LIN {X 0,Y 411.212,Z 369.263,A -85,B 0,C 180,E1 -10675.122,E2 -10675.122} C_VEL
LIN {X 0,Y 411.168,Z 369.267,A -85,B 0,C 180,E1 -10678.003,E2 -10678.003} C_VEL
LIN {X 0,Y 411.22,Z 369.26,A -85,B 0,C 180,E1 -10681.41,E2 -10681.41} C_VEL
LIN {X 0,Y 411.24,Z 369.258,A -85,B 0,C 180,E1 -10683.619,E2 -10683.619} C_VEL
LIN {X 0,Y 411.205,Z 369.264,A -85,B 0,C 180,E1 -10686.853,E2 -10686.853} C_VEL
LIN {X 0,Y 411.267,Z 369.256,A -85,B 0,C 180,E1 -10690.031,E2 -10690.031} C_VEL
LIN {X 0,Y 411.267,Z 369.255,A -85,B 0,C 180,E1 -10693.131,E2 -10693.131} C_VEL
LIN {X 0,Y 411.308,Z 369.251,A -85,B 0,C 180,E1 -10696.896,E2 -10696.896} C_VEL
LIN {X 0,Y 411.307,Z 369.253,A -85,B 0,C 180,E1 -10700.162,E2 -10700.162} C_VEL
LIN {X 0,Y 411.455,Z 369.23,A -85,B 0,C 180,E1 -10703.133,E2 -10703.133} C_VEL
LIN {X 0,Y 411.313,Z 369.249,A -85,B 0,C 180,E1 -10705.099,E2 -10705.099} C_VEL
LIN {X 0,Y 411.515,Z 369.226,A -85,B 0,C 180,E1 -10708.043,E2 -10708.043} C_VEL
LIN {X 0,Y 411.646,Z 369.21,A -85,B 0,C 180,E1 -10710,E2 -10710} C_VEL
LIN {X 0,Y 411.461,Z 369.229,A -85,B 0,C 180,E1 -10712.937,E2 -10712.937} C_VEL
LIN {X 0,Y 411.455,Z 369.232,A -85,B 0,C 180,E1 -10716.867,E2 -10716.867} C_VEL
LIN {X 0,Y 411.297,Z 369.253,A -85,B 0,C 180,E1 -10719.839,E2 -10719.839} C_VEL
LIN {X 0,Y 411.287,Z 369.252,A -85,B 0,C 180,E1 -10723.319,E2 -10723.319} C_VEL
LIN {X 0,Y 411.26,Z 369.256,A -85,B 0,C 180,E1 -10726.889,E2 -10726.889} C_VEL
LIN {X 0,Y 411.243,Z 369.257,A -85,B 0,C 180,E1 -10727.585,E2 -10727.585} C_VEL
LIN {X 0,Y 410.582,Z 369.343,A -85,B 0,C 180,E1 -10728.403,E2 -10728.403} C_VEL
LIN {X 0,Y 407.695,Z 369.704,A -85,B 0,C 180,E1 -10729.731,E2 -10729.731} C_VEL
LIN {X 0,Y 405.251,Z 370.006,A -85,B 0,C 180,E1 -10730.804,E2 -10730.804} C_VEL
LIN {X 0,Y 404.215,Z 370.136,A -85,B 0,C 180,E1 -10731.634,E2 -10731.634} C_VEL
LIN {X 0,Y 404.139,Z 370.141,A -85,B 0,C 180,E1 -10731.915,E2 -10731.915} C_VEL
LIN {X 0,Y 404.219,Z 370.134,A -85,B 0,C 180,E1 -10735.297,E2 -10735.297} C_VEL
LIN {X 0,Y 404.198,Z 370.137,A -85,B 0,C 180,E1 -10738,E2 -10738} C_VEL
LIN {X 0,Y 404.142,Z 370.145,A -85,B 0,C 180,E1 -10741.558,E2 -10741.558} C_VEL
LIN {X 0,Y 404.187,Z 370.137,A -85,B 0,C 180,E1 -10745.016,E2 -10745.016} C_VEL
LIN {X 0,Y 404.159,Z 370.141,A -85,B 0,C 180,E1 -10748.757,E2 -10748.757} C_VEL
LIN {X 0,Y 404.127,Z 370.147,A -85,B 0,C 180,E1 -10751.6,E2 -10751.6} C_VEL
LIN {X 0,Y 404.151,Z 370.141,A -85,B 0,C 180,E1 -10754.523,E2 -10754.523} C_VEL
LIN {X 0,Y 404.139,Z 370.146,A -85,B 0,C 180,E1 -10757.296,E2 -10757.296} C_VEL
LIN {X 0,Y 404.172,Z 370.139,A -85,B 0,C 180,E1 -10759.955,E2 -10759.955} C_VEL
LIN {X 0,Y 404.143,Z 370.144,A -85,B 0,C 180,E1 -10763.124,E2 -10763.124} C_VEL
LIN {X 0,Y 404.149,Z 370.141,A -85,B 0,C 180,E1 -10766.188,E2 -10766.188} C_VEL
LIN {X 0,Y 404.345,Z 370.296,A -85,B 0,C 180,E1 -10769.153,E2 -10769.153} C_VEL
LIN {X 0,Y 404.32,Z 374.446,A -85,B 0,C 180,E1 -10771.444,E2 -10771.444} C_VEL
LIN {X 0,Y 404.015,Z 380.585,A -85,B 0,C 180,E1 -10774.765,E2 -10774.765} C_VEL
LIN {X 0,Y 403.792,Z 386.695,A -85,B 0,C 180,E1 -10778.025,E2 -10778.025} C_VEL
LIN {X 0,Y 403.633,Z 392.803,A -85,B 0,C 180,E1 -10781.209,E2 -10781.209} C_VEL
LIN {X 0,Y 403.511,Z 398.878,A -85,B 0,C 180,E1 -10784.338,E2 -10784.338} C_VEL
LIN {X 0,Y 403.32,Z 405.986,A -85,B 0,C 180,E1 -10787.93,E2 -10787.93} C_VEL
LIN {X 0,Y 403.258,Z 409.014,A -85,B 0,C 180,E1 -10789.424,E2 -10789.424} C_VEL
LIN {X 0,Y 404.669,Z 419.398,A -85,B 0,C 180,E1 -10789.999,E2 -10789.999} C_VEL
LIN {X 0,Y 405.097,Z 425.037,A -85,B 0,C 180,E1 -10790.387,E2 -10790.387} C_VEL
LIN {X 0,Y 404.722,Z 435.358,A -85,B 0,C 180,E1 -10791.26,E2 -10791.26} C_VEL
LIN {X 0,Y 404.281,Z 444.367,A -85,B 0,C 180,E1 -10792.261,E2 -10792.261} C_VEL
LIN {X 0,Y 404.112,Z 451.373,A -85,B 0,C 180,E1 -10793.258,E2 -10793.258} C_VEL
LIN {X 0,Y 403.938,Z 458.258,A -85,B 0,C 180,E1 -10794.509,E2 -10794.509} C_VEL
LIN {X 0,Y 403.774,Z 462.57,A -85,B 0,C 180,E1 -10795.508,E2 -10795.508} C_VEL
LIN {X 0,Y 403.609,Z 465.969,A -85,B 0,C 180,E1 -10796.506,E2 -10796.506} C_VEL
LIN {X 0,Y 403.281,Z 469.606,A -85,B 0,C 180,E1 -10798.003,E2 -10798.003} C_VEL
LIN {X 0,Y 403.192,Z 471.134,A -85,B 0,C 180,E1 -10799.001,E2 -10799.001} C_VEL
LIN {X 0,Y 403.19,Z 471.985,A -85,B 0,C 180,E1 -10800,E2 -10800} C_VEL
LIN {X 0,Y 403.247,Z 472.168,A -85,B 0,C 180,E1 -10800.999,E2 -10800.999} C_VEL
LIN {X 0,Y 403.356,Z 471.686,A -85,B 0,C 180,E1 -10801.997,E2 -10801.997} C_VEL
LIN {X 0,Y 403.54,Z 470.533,A -85,B 0,C 180,E1 -10802.995,E2 -10802.995} C_VEL
LIN {X 0,Y 404.138,Z 467.465,A -85,B 0,C 180,E1 -10804.488,E2 -10804.488} C_VEL
LIN {X 0,Y 404.326,Z 464.514,A -85,B 0,C 180,E1 -10805.486,E2 -10805.486} C_VEL
LIN {X 0,Y 404.807,Z 459.63,A -85,B 0,C 180,E1 -10806.73,E2 -10806.73} C_VEL
LIN {X 0,Y 405.372,Z 453.215,A -85,B 0,C 180,E1 -10807.972,E2 -10807.972} C_VEL
LIN {X 0,Y 405.95,Z 446.675,A -85,B 0,C 180,E1 -10808.964,E2 -10808.964} C_VEL
LIN {X 0,Y 406.576,Z 438.47,A -85,B 0,C 180,E1 -10809.954,E2 -10809.954} C_VEL
LIN {X 0,Y 407.173,Z 429.296,A -85,B 0,C 180,E1 -10810.819,E2 -10810.819} C_VEL
LIN {X 0,Y 406.43,Z 423.17,A -85,B 0,C 180,E1 -10811.344,E2 -10811.344} C_VEL
LIN {X 0,Y 404.018,Z 412.539,A -85,B 0,C 180,E1 -10812.176,E2 -10812.176} C_VEL
LIN {X 0,Y 404.254,Z 407.353,A -85,B 0,C 180,E1 -10815.116,E2 -10815.116} C_VEL
LIN {X 0,Y 404.598,Z 402.059,A -85,B 0,C 180,E1 -10818.22,E2 -10818.22} C_VEL
LIN {X 0,Y 404.945,Z 396.896,A -85,B 0,C 180,E1 -10821.375,E2 -10821.375} C_VEL
LIN {X 0,Y 405.44,Z 391.905,A -85,B 0,C 180,E1 -10824.584,E2 -10824.584} C_VEL
LIN {X 0,Y 406.072,Z 386.86,A -85,B 0,C 180,E1 -10828.033,E2 -10828.033} C_VEL
LIN {X 0,Y 406.384,Z 384.059,A -85,B 0,C 180,E1 -10830.151,E2 -10830.151} C_VEL
LIN {X 0,Y 406.317,Z 381.396,A -85,B 0,C 180,E1 -10832.426,E2 -10832.426} C_VEL
LIN {X 0,Y 406.022,Z 379.03,A -85,B 0,C 180,E1 -10834.835,E2 -10834.835} C_VEL
LIN {X 0,Y 405.683,Z 377.136,A -85,B 0,C 180,E1 -10837.325,E2 -10837.325} C_VEL
LIN {X 0,Y 405.446,Z 375.637,A -85,B 0,C 180,E1 -10840.297,E2 -10840.297} C_VEL
LIN {X 0,Y 405.397,Z 375.192,A -85,B 0,C 180,E1 -10843.271,E2 -10843.271} C_VEL
LIN {X 0,Y 405.551,Z 375.903,A -85,B 0,C 180,E1 -10846.117,E2 -10846.117} C_VEL
LIN {X 0,Y 406.076,Z 377.767,A -85,B 0,C 180,E1 -10848.877,E2 -10848.877} C_VEL
LIN {X 0,Y 406.772,Z 380.667,A -85,B 0,C 180,E1 -10851.538,E2 -10851.538} C_VEL
LIN {X 0,Y 408.037,Z 385.656,A -85,B 0,C 180,E1 -10854.76,E2 -10854.76} C_VEL
LIN {X 0,Y 409.173,Z 390.814,A -85,B 0,C 180,E1 -10857.313,E2 -10857.313} C_VEL
LIN {X 0,Y 410.133,Z 396.458,A -85,B 0,C 180,E1 -10859.635,E2 -10859.635} C_VEL
LIN {X 0,Y 409.985,Z 399.501,A -85,B 0,C 180,E1 -10860.695,E2 -10860.695} C_VEL
LIN {X 0,Y 407.911,Z 410.385,A -85,B 0,C 180,E1 -10864.008,E2 -10864.008} C_VEL
LIN {X 0,Y 406.44,Z 421.407,A -85,B 0,C 180,E1 -10867.104,E2 -10867.104} C_VEL
LIN {X 0,Y 405.209,Z 434.333,A -85,B 0,C 180,E1 -10870.496,E2 -10870.496} C_VEL
LIN {X 0,Y 404.648,Z 442.082,A -85,B 0,C 180,E1 -10872.397,E2 -10872.397} C_VEL
LIN {X 0,Y 406.509,Z 454.809,A -85,B 0,C 180,E1 -10872.908,E2 -10872.908} C_VEL
LIN {X 0,Y 407.267,Z 468.253,A -85,B 0,C 180,E1 -10873.601,E2 -10873.601} C_VEL
LIN {X 0,Y 406.773,Z 479.668,A -85,B 0,C 180,E1 -10874.338,E2 -10874.338} C_VEL
LIN {X 0,Y 405.87,Z 491.757,A -85,B 0,C 180,E1 -10875.33,E2 -10875.33} C_VEL
LIN {X 0,Y 405.11,Z 502.511,A -85,B 0,C 180,E1 -10876.462,E2 -10876.462} C_VEL
LIN {X 0,Y 404.391,Z 512.142,A -85,B 0,C 180,E1 -10877.708,E2 -10877.708} C_VEL
LIN {X 0,Y 403.888,Z 520.09,A -85,B 0,C 180,E1 -10878.965,E2 -10878.965} C_VEL
LIN {X 0,Y 403.457,Z 527.841,A -85,B 0,C 180,E1 -10880.474,E2 -10880.474} C_VEL
LIN {X 0,Y 403.222,Z 534.087,A -85,B 0,C 180,E1 -10881.985,E2 -10881.985} C_VEL
LIN {X 0,Y 403.136,Z 539.248,A -85,B 0,C 180,E1 -10883.567,E2 -10883.567} C_VEL
LIN {X 0,Y 403.096,Z 542.795,A -85,B 0,C 180,E1 -10884.999,E2 -10884.999} C_VEL
LIN {X 0,Y 403.113,Z 544.709,A -85,B 0,C 180,E1 -10886.001,E2 -10886.001} C_VEL
LIN {X 0,Y 403.202,Z 546.163,A -85,B 0,C 180,E1 -10887.002,E2 -10887.002} C_VEL
LIN {X 0,Y 403.218,Z 547.195,A -85,B 0,C 180,E1 -10888.002,E2 -10888.002} C_VEL
LIN {X 0,Y 403.123,Z 547.774,A -85,B 0,C 180,E1 -10889.001,E2 -10889.001} C_VEL
LIN {X 0,Y 403.102,Z 547.905,A -85,B 0,C 180,E1 -10890,E2 -10890} C_VEL
LIN {X 0,Y 403.121,Z 547.631,A -85,B 0,C 180,E1 -10890.999,E2 -10890.999} C_VEL
LIN {X 0,Y 403.223,Z 546.941,A -85,B 0,C 180,E1 -10891.997,E2 -10891.997} C_VEL
LIN {X 0,Y 403.268,Z 545.766,A -85,B 0,C 180,E1 -10892.997,E2 -10892.997} C_VEL
LIN {X 0,Y 403.099,Z 543.145,A -85,B 0,C 180,E1 -10894.5,E2 -10894.5} C_VEL
LIN {X 0,Y 403.142,Z 539.441,A -85,B 0,C 180,E1 -10896.004,E2 -10896.004} C_VEL
LIN {X 0,Y 403.201,Z 534.528,A -85,B 0,C 180,E1 -10897.512,E2 -10897.512} C_VEL
LIN {X 0,Y 403.358,Z 528.258,A -85,B 0,C 180,E1 -10899.022,E2 -10899.022} C_VEL
LIN {X 0,Y 403.681,Z 520.298,A -85,B 0,C 180,E1 -10900.533,E2 -10900.533} C_VEL
LIN {X 0,Y 404.134,Z 512.119,A -85,B 0,C 180,E1 -10901.79,E2 -10901.79} C_VEL
LIN {X 0,Y 404.728,Z 502.074,A -85,B 0,C 180,E1 -10903.046,E2 -10903.046} C_VEL
LIN {X 0,Y 405.281,Z 492.039,A -85,B 0,C 180,E1 -10904.05,E2 -10904.05} C_VEL
LIN {X 0,Y 405.86,Z 481.103,A -85,B 0,C 180,E1 -10904.926,E2 -10904.926} C_VEL
LIN {X 0,Y 406.416,Z 468.992,A -85,B 0,C 180,E1 -10905.676,E2 -10905.676} C_VEL
LIN {X 0,Y 405.399,Z 456.125,A -85,B 0,C 180,E1 -10906.276,E2 -10906.276} C_VEL
LIN {X 0,Y 404.221,Z 443.249,A -85,B 0,C 180,E1 -10906.7,E2 -10906.7} C_VEL
LIN {X 0,Y 405.015,Z 430.654,A -85,B 0,C 180,E1 -10909.778,E2 -10909.778} C_VEL
LIN {X 0,Y 406.134,Z 416.925,A -85,B 0,C 180,E1 -10913.184,E2 -10913.184} C_VEL
LIN {X 0,Y 407.489,Z 403.197,A -85,B 0,C 180,E1 -10916.642,E2 -10916.642} C_VEL
LIN {X 0,Y 408.621,Z 392.664,A -85,B 0,C 180,E1 -10919.352,E2 -10919.352} C_VEL
LIN {X 0,Y 407.859,Z 387.494,A -85,B 0,C 180,E1 -10920.778,E2 -10920.778} C_VEL
LIN {X 0,Y 405.306,Z 375.4,A -85,B 0,C 180,E1 -10924.301,E2 -10924.301} C_VEL
LIN {X 0,Y 404.175,Z 370.14,A -85,B 0,C 180,E1 -10925.906,E2 -10925.906} C_VEL
LIN {X 0,Y 404.155,Z 370.141,A -85,B 0,C 180,E1 -10928.757,E2 -10928.757} C_VEL
LIN {X 0,Y 404.125,Z 370.148,A -85,B 0,C 180,E1 -10931.6,E2 -10931.6} C_VEL
LIN {X 0,Y 404.151,Z 370.143,A -85,B 0,C 180,E1 -10934.523,E2 -10934.523} C_VEL
LIN {X 0,Y 404.141,Z 370.142,A -85,B 0,C 180,E1 -10937.296,E2 -10937.296} C_VEL
LIN {X 0,Y 404.169,Z 370.141,A -85,B 0,C 180,E1 -10939.955,E2 -10939.955} C_VEL
LIN {X 0,Y 404.141,Z 370.142,A -85,B 0,C 180,E1 -10943.124,E2 -10943.124} C_VEL
LIN {X 0,Y 404.146,Z 370.144,A -85,B 0,C 180,E1 -10946.188,E2 -10946.188} C_VEL
LIN {X 0,Y 404.146,Z 370.143,A -85,B 0,C 180,E1 -10949.715,E2 -10949.715} C_VEL
LIN {X 0,Y 404.196,Z 370.135,A -85,B 0,C 180,E1 -10953.123,E2 -10953.123} C_VEL
LIN {X 0,Y 404.178,Z 370.139,A -85,B 0,C 180,E1 -10955.334,E2 -10955.334} C_VEL
LIN {X 0,Y 404.14,Z 370.143,A -85,B 0,C 180,E1 -10958.581,E2 -10958.581} C_VEL
LIN {X 0,Y 404.211,Z 370.137,A -85,B 0,C 180,E1 -10961.762,E2 -10961.762} C_VEL
LIN {X 0,Y 404.208,Z 370.134,A -85,B 0,C 180,E1 -10964.882,E2 -10964.882} C_VEL
LIN {X 0,Y 404.258,Z 370.13,A -85,B 0,C 180,E1 -10967.959,E2 -10967.959} C_VEL
LIN {X 0,Y 404.434,Z 370.106,A -85,B 0,C 180,E1 -10972.1,E2 -10972.1} C_VEL
LIN {X 0,Y 404.425,Z 370.108,A -85,B 0,C 180,E1 -10974.015,E2 -10974.015} C_VEL
LIN {X 0,Y 404.484,Z 370.102,A -85,B 0,C 180,E1 -10978.009,E2 -10978.009} C_VEL
LIN {X 0,Y 404.613,Z 370.085,A -85,B 0,C 180,E1 -10980,E2 -10980} C_VEL
LIN {X 0,Y 404.417,Z 370.108,A -85,B 0,C 180,E1 -10982.988,E2 -10982.988} C_VEL
LIN {X 0,Y 404.413,Z 370.11,A -85,B 0,C 180,E1 -10986.987,E2 -10986.987} C_VEL
LIN {X 0,Y 404.272,Z 370.127,A -85,B 0,C 180,E1 -10990.011,E2 -10990.011} C_VEL
LIN {X 0,Y 404.267,Z 370.129,A -85,B 0,C 180,E1 -10993.211,E2 -10993.211} C_VEL
LIN {X 0,Y 404.217,Z 370.136,A -85,B 0,C 180,E1 -10997.007,E2 -10997.007} C_VEL
LIN {X 0,Y 404.165,Z 370.14,A -85,B 0,C 180,E1 -11000.352,E2 -11000.352} C_VEL
LIN {X 0,Y 404.171,Z 370.14,A -85,B 0,C 180,E1 -11003.575,E2 -11003.575} C_VEL
LIN {X 0,Y 404.185,Z 370.136,A -85,B 0,C 180,E1 -11005.766,E2 -11005.766} C_VEL
LIN {X 0,Y 404.196,Z 370.135,A -85,B 0,C 180,E1 -11008,E2 -11008} C_VEL
LIN {X 0,Y 404.14,Z 370.144,A -85,B 0,C 180,E1 -11011.558,E2 -11011.558} C_VEL
LIN {X 0,Y 404.187,Z 370.14,A -85,B 0,C 180,E1 -11015.016,E2 -11015.016} C_VEL
LIN {X 0,Y 404.158,Z 370.145,A -85,B 0,C 180,E1 -11018.757,E2 -11018.757} C_VEL
LIN {X 0,Y 404.124,Z 370.145,A -85,B 0,C 180,E1 -11021.6,E2 -11021.6} C_VEL
LIN {X 0,Y 404.148,Z 370.143,A -85,B 0,C 180,E1 -11024.522,E2 -11024.522} C_VEL
LIN {X 0,Y 404.141,Z 370.142,A -85,B 0,C 180,E1 -11027.296,E2 -11027.296} C_VEL
LIN {X 0,Y 404.17,Z 370.138,A -85,B 0,C 180,E1 -11029.956,E2 -11029.956} C_VEL
LIN {X 0,Y 404.138,Z 370.145,A -85,B 0,C 180,E1 -11033.125,E2 -11033.125} C_VEL
LIN {X 0,Y 404.146,Z 370.143,A -85,B 0,C 180,E1 -11036.188,E2 -11036.188} C_VEL
LIN {X 0,Y 404.147,Z 370.14,A -85,B 0,C 180,E1 -11039.715,E2 -11039.715} C_VEL
LIN {X 0,Y 404.197,Z 370.136,A -85,B 0,C 180,E1 -11043.123,E2 -11043.123} C_VEL
LIN {X 0,Y 404.179,Z 370.138,A -85,B 0,C 180,E1 -11045.335,E2 -11045.335} C_VEL
LIN {X 0,Y 404.165,Z 370.143,A -85,B 0,C 180,E1 -11048.582,E2 -11048.582} C_VEL
LIN {X 0,Y 404.217,Z 370.133,A -85,B 0,C 180,E1 -11051.762,E2 -11051.762} C_VEL
LIN {X 0,Y 404.214,Z 370.134,A -85,B 0,C 180,E1 -11054.882,E2 -11054.882} C_VEL
LIN {X 0,Y 404.259,Z 370.129,A -85,B 0,C 180,E1 -11057.959,E2 -11057.959} C_VEL
LIN {X 0,Y 404.386,Z 370.115,A -85,B 0,C 180,E1 -11062.008,E2 -11062.008} C_VEL
LIN {X 0,Y 404.422,Z 370.111,A -85,B 0,C 180,E1 -11064.015,E2 -11064.015} C_VEL
LIN {X 0,Y 404.484,Z 370.102,A -85,B 0,C 180,E1 -11068.009,E2 -11068.009} C_VEL
LIN {X 0,Y 404.615,Z 370.086,A -85,B 0,C 180,E1 -11070,E2 -11070} C_VEL
LIN {X 0,Y 404.419,Z 370.106,A -85,B 0,C 180,E1 -11072.989,E2 -11072.989} C_VEL
LIN {X 0,Y 404.422,Z 370.109,A -85,B 0,C 180,E1 -11075.985,E2 -11075.985} C_VEL
LIN {X 0,Y 404.295,Z 370.124,A -85,B 0,C 180,E1 -11079.001,E2 -11079.001} C_VEL
LIN {X 0,Y 404.26,Z 370.13,A -85,B 0,C 180,E1 -11082.042,E2 -11082.042} C_VEL
LIN {X 0,Y 404.21,Z 370.134,A -85,B 0,C 180,E1 -11085.118,E2 -11085.118} C_VEL
LIN {X 0,Y 404.213,Z 370.135,A -85,B 0,C 180,E1 -11088.238,E2 -11088.238} C_VEL
LIN {X 0,Y 404.142,Z 370.144,A -85,B 0,C 180,E1 -11091.419,E2 -11091.419} C_VEL
LIN {X 0,Y 404.139,Z 370.141,A -85,B 0,C 180,E1 -11091.915,E2 -11091.915} C_VEL
LIN {X 0,Y 403.496,Z 370.223,A -85,B 0,C 180,E1 -11092.746,E2 -11092.746} C_VEL
LIN {X 0,Y 400.664,Z 370.576,A -85,B 0,C 180,E1 -11094.098,E2 -11094.098} C_VEL
LIN {X 0,Y 398.254,Z 370.877,A -85,B 0,C 180,E1 -11095.19,E2 -11095.19} C_VEL
LIN {X 0,Y 397.22,Z 371.005,A -85,B 0,C 180,E1 -11096.034,E2 -11096.034} C_VEL
LIN {X 0,Y 397.137,Z 371.014,A -85,B 0,C 180,E1 -11096.32,E2 -11096.32} C_VEL
LIN {X 0,Y 397.125,Z 371.016,A -85,B 0,C 180,E1 -11098.544,E2 -11098.544} C_VEL
LIN {X 0,Y 397.081,Z 371.023,A -85,B 0,C 180,E1 -11102.072,E2 -11102.072} C_VEL
LIN {X 0,Y 397.122,Z 371.02,A -85,B 0,C 180,E1 -11105.503,E2 -11105.503} C_VEL
LIN {X 0,Y 397.134,Z 371.017,A -85,B 0,C 180,E1 -11108.862,E2 -11108.862} C_VEL
LIN {X 0,Y 397.074,Z 371.023,A -85,B 0,C 180,E1 -11112.267,E2 -11112.267} C_VEL
LIN {X 0,Y 397.092,Z 371.022,A -85,B 0,C 180,E1 -11115.069,E2 -11115.069} C_VEL
LIN {X 0,Y 397.069,Z 371.022,A -85,B 0,C 180,E1 -11118.021,E2 -11118.021} C_VEL
LIN {X 0,Y 397.136,Z 371.017,A -85,B 0,C 180,E1 -11121.138,E2 -11121.138} C_VEL
LIN {X 0,Y 397.123,Z 371.017,A -85,B 0,C 180,E1 -11124.497,E2 -11124.497} C_VEL
LIN {X 0,Y 397.164,Z 371.013,A -85,B 0,C 180,E1 -11128.145,E2 -11128.145} C_VEL
LIN {X 0,Y 397.291,Z 371.125,A -85,B 0,C 180,E1 -11129.062,E2 -11129.062} C_VEL
LIN {X 0,Y 397.323,Z 374.396,A -85,B 0,C 180,E1 -11130.894,E2 -11130.894} C_VEL
LIN {X 0,Y 396.973,Z 381.037,A -85,B 0,C 180,E1 -11134.543,E2 -11134.543} C_VEL
LIN {X 0,Y 396.763,Z 386.773,A -85,B 0,C 180,E1 -11137.621,E2 -11137.621} C_VEL
LIN {X 0,Y 396.589,Z 392.898,A -85,B 0,C 180,E1 -11140.862,E2 -11140.862} C_VEL
LIN {X 0,Y 396.448,Z 399,A -85,B 0,C 180,E1 -11144.051,E2 -11144.051} C_VEL
LIN {X 0,Y 396.272,Z 406.161,A -85,B 0,C 180,E1 -11147.712,E2 -11147.712} C_VEL
LIN {X 0,Y 396.16,Z 409.279,A -85,B 0,C 180,E1 -11149.265,E2 -11149.265} C_VEL
LIN {X 0,Y 397.641,Z 420.176,A -85,B 0,C 180,E1 -11149.884,E2 -11149.884} C_VEL
LIN {X 0,Y 398.045,Z 426.586,A -85,B 0,C 180,E1 -11150.344,E2 -11150.344} C_VEL
LIN {X 0,Y 397.651,Z 436.659,A -85,B 0,C 180,E1 -11151.232,E2 -11151.232} C_VEL
LIN {X 0,Y 397.231,Z 445.211,A -85,B 0,C 180,E1 -11152.215,E2 -11152.215} C_VEL
LIN {X 0,Y 397.057,Z 453.143,A -85,B 0,C 180,E1 -11153.393,E2 -11153.393} C_VEL
LIN {X 0,Y 396.838,Z 459.749,A -85,B 0,C 180,E1 -11154.665,E2 -11154.665} C_VEL
LIN {X 0,Y 396.593,Z 464.783,A -85,B 0,C 180,E1 -11155.935,E2 -11155.935} C_VEL
LIN {X 0,Y 396.36,Z 467.853,A -85,B 0,C 180,E1 -11156.951,E2 -11156.951} C_VEL
LIN {X 0,Y 396.233,Z 470.158,A -85,B 0,C 180,E1 -11157.967,E2 -11157.967} C_VEL
LIN {X 0,Y 396.136,Z 471.757,A -85,B 0,C 180,E1 -11158.983,E2 -11158.983} C_VEL
LIN {X 0,Y 396.13,Z 472.676,A -85,B 0,C 180,E1 -11160,E2 -11160} C_VEL
LIN {X 0,Y 396.189,Z 472.923,A -85,B 0,C 180,E1 -11161.016,E2 -11161.016} C_VEL
LIN {X 0,Y 396.309,Z 472.502,A -85,B 0,C 180,E1 -11162.033,E2 -11162.033} C_VEL
LIN {X 0,Y 396.505,Z 471.41,A -85,B 0,C 180,E1 -11163.048,E2 -11163.048} C_VEL
LIN {X 0,Y 397.127,Z 468.457,A -85,B 0,C 180,E1 -11164.568,E2 -11164.568} C_VEL
LIN {X 0,Y 397.365,Z 465.61,A -85,B 0,C 180,E1 -11165.582,E2 -11165.582} C_VEL
LIN {X 0,Y 397.876,Z 460.871,A -85,B 0,C 180,E1 -11166.848,E2 -11166.848} C_VEL
LIN {X 0,Y 398.461,Z 454.631,A -85,B 0,C 180,E1 -11168.112,E2 -11168.112} C_VEL
LIN {X 0,Y 399.216,Z 446.466,A -85,B 0,C 180,E1 -11169.372,E2 -11169.372} C_VEL
LIN {X 0,Y 399.932,Z 438.019,A -85,B 0,C 180,E1 -11170.377,E2 -11170.377} C_VEL
LIN {X 0,Y 400.41,Z 428.651,A -85,B 0,C 180,E1 -11171.26,E2 -11171.26} C_VEL
LIN {X 0,Y 398.605,Z 419.229,A -85,B 0,C 180,E1 -11172.086,E2 -11172.086} C_VEL
LIN {X 0,Y 397.088,Z 413.056,A -85,B 0,C 180,E1 -11172.57,E2 -11172.57} C_VEL
LIN {X 0,Y 397.396,Z 406.452,A -85,B 0,C 180,E1 -11176.437,E2 -11176.437} C_VEL
LIN {X 0,Y 397.787,Z 401.229,A -85,B 0,C 180,E1 -11179.614,E2 -11179.614} C_VEL
LIN {X 0,Y 398.332,Z 395.288,A -85,B 0,C 180,E1 -11183.441,E2 -11183.441} C_VEL
LIN {X 0,Y 399.018,Z 389.746,A -85,B 0,C 180,E1 -11187.255,E2 -11187.255} C_VEL
LIN {X 0,Y 399.437,Z 386.761,A -85,B 0,C 180,E1 -11189.515,E2 -11189.515} C_VEL
LIN {X 0,Y 399.538,Z 383.439,A -85,B 0,C 180,E1 -11192.399,E2 -11192.399} C_VEL
LIN {X 0,Y 399.185,Z 380.624,A -85,B 0,C 180,E1 -11195.521,E2 -11195.521} C_VEL
LIN {X 0,Y 398.822,Z 378.445,A -85,B 0,C 180,E1 -11199.162,E2 -11199.162} C_VEL
LIN {X 0,Y 398.721,Z 377.703,A -85,B 0,C 180,E1 -11202.052,E2 -11202.052} C_VEL
LIN {X 0,Y 398.827,Z 378.008,A -85,B 0,C 180,E1 -11204.819,E2 -11204.819} C_VEL
LIN {X 0,Y 399.213,Z 379.398,A -85,B 0,C 180,E1 -11207.68,E2 -11207.68} C_VEL
LIN {X 0,Y 399.88,Z 382.14,A -85,B 0,C 180,E1 -11210.652,E2 -11210.652} C_VEL
LIN {X 0,Y 400.749,Z 385.848,A -85,B 0,C 180,E1 -11213.397,E2 -11213.397} C_VEL
LIN {X 0,Y 401.642,Z 389.151,A -85,B 0,C 180,E1 -11215.327,E2 -11215.327} C_VEL
LIN {X 0,Y 402.693,Z 394.363,A -85,B 0,C 180,E1 -11217.839,E2 -11217.839} C_VEL
LIN {X 0,Y 403.354,Z 398.737,A -85,B 0,C 180,E1 -11219.649,E2 -11219.649} C_VEL
LIN {X 0,Y 403.051,Z 401.938,A -85,B 0,C 180,E1 -11220.775,E2 -11220.775} C_VEL
LIN {X 0,Y 400.978,Z 412.337,A -85,B 0,C 180,E1 -11224.012,E2 -11224.012} C_VEL
LIN {X 0,Y 399.404,Z 423.52,A -85,B 0,C 180,E1 -11227.225,E2 -11227.225} C_VEL
LIN {X 0,Y 398.15,Z 436.391,A -85,B 0,C 180,E1 -11230.672,E2 -11230.672} C_VEL
LIN {X 0,Y 397.711,Z 441.528,A -85,B 0,C 180,E1 -11231.993,E2 -11231.993} C_VEL
LIN {X 0,Y 399.636,Z 454.304,A -85,B 0,C 180,E1 -11232.535,E2 -11232.535} C_VEL
LIN {X 0,Y 400.372,Z 467.262,A -85,B 0,C 180,E1 -11233.221,E2 -11233.221} C_VEL
LIN {X 0,Y 400.317,Z 474.503,A -85,B 0,C 180,E1 -11233.686,E2 -11233.686} C_VEL
LIN {X 0,Y 399.431,Z 486.15,A -85,B 0,C 180,E1 -11234.566,E2 -11234.566} C_VEL
LIN {X 0,Y 398.632,Z 496.658,A -85,B 0,C 180,E1 -11235.58,E2 -11235.58} C_VEL
LIN {X 0,Y 397.908,Z 506.32,A -85,B 0,C 180,E1 -11236.726,E2 -11236.726} C_VEL
LIN {X 0,Y 397.187,Z 515.15,A -85,B 0,C 180,E1 -11238,E2 -11238} C_VEL
LIN {X 0,Y 396.564,Z 523.737,A -85,B 0,C 180,E1 -11239.534,E2 -11239.534} C_VEL
LIN {X 0,Y 396.259,Z 530.655,A -85,B 0,C 180,E1 -11241.072,E2 -11241.072} C_VEL
LIN {X 0,Y 396.095,Z 536.981,A -85,B 0,C 180,E1 -11242.865,E2 -11242.865} C_VEL
LIN {X 0,Y 396.029,Z 541.076,A -85,B 0,C 180,E1 -11244.399,E2 -11244.399} C_VEL
LIN {X 0,Y 396.023,Z 544.085,A -85,B 0,C 180,E1 -11245.929,E2 -11245.929} C_VEL
LIN {X 0,Y 396.13,Z 545.524,A -85,B 0,C 180,E1 -11246.949,E2 -11246.949} C_VEL
LIN {X 0,Y 396.167,Z 546.542,A -85,B 0,C 180,E1 -11247.967,E2 -11247.967} C_VEL
LIN {X 0,Y 396.071,Z 547.083,A -85,B 0,C 180,E1 -11248.983,E2 -11248.983} C_VEL
LIN {X 0,Y 396.047,Z 547.197,A -85,B 0,C 180,E1 -11250,E2 -11250} C_VEL
LIN {X 0,Y 396.07,Z 546.905,A -85,B 0,C 180,E1 -11251.017,E2 -11251.017} C_VEL
LIN {X 0,Y 396.175,Z 546.172,A -85,B 0,C 180,E1 -11252.033,E2 -11252.033} C_VEL
LIN {X 0,Y 396.193,Z 544.97,A -85,B 0,C 180,E1 -11253.05,E2 -11253.05} C_VEL
LIN {X 0,Y 396.026,Z 542.296,A -85,B 0,C 180,E1 -11254.58,E2 -11254.58} C_VEL
LIN {X 0,Y 396.085,Z 538.534,A -85,B 0,C 180,E1 -11256.111,E2 -11256.111} C_VEL
LIN {X 0,Y 396.145,Z 533.552,A -85,B 0,C 180,E1 -11257.646,E2 -11257.646} C_VEL
LIN {X 0,Y 396.311,Z 527.179,A -85,B 0,C 180,E1 -11259.184,E2 -11259.184} C_VEL
LIN {X 0,Y 396.657,Z 519.098,A -85,B 0,C 180,E1 -11260.722,E2 -11260.722} C_VEL
LIN {X 0,Y 397.08,Z 510.792,A -85,B 0,C 180,E1 -11262.003,E2 -11262.003} C_VEL
LIN {X 0,Y 397.657,Z 501.686,A -85,B 0,C 180,E1 -11263.152,E2 -11263.152} C_VEL
LIN {X 0,Y 398.27,Z 491.511,A -85,B 0,C 180,E1 -11264.19,E2 -11264.19} C_VEL
LIN {X 0,Y 398.844,Z 480.816,A -85,B 0,C 180,E1 -11265.064,E2 -11265.064} C_VEL
LIN {X 0,Y 399.366,Z 468.773,A -85,B 0,C 180,E1 -11265.829,E2 -11265.829} C_VEL
LIN {X 0,Y 398.31,Z 455.912,A -85,B 0,C 180,E1 -11266.446,E2 -11266.446} C_VEL
LIN {X 0,Y 397.173,Z 442.976,A -85,B 0,C 180,E1 -11266.879,E2 -11266.879} C_VEL
LIN {X 0,Y 397.959,Z 431.03,A -85,B 0,C 180,E1 -11269.874,E2 -11269.874} C_VEL
LIN {X 0,Y 399.107,Z 417.627,A -85,B 0,C 180,E1 -11273.278,E2 -11273.278} C_VEL
LIN {X 0,Y 400.497,Z 404.176,A -85,B 0,C 180,E1 -11276.733,E2 -11276.733} C_VEL
LIN {X 0,Y 401.632,Z 394.243,A -85,B 0,C 180,E1 -11279.338,E2 -11279.338} C_VEL
LIN {X 0,Y 401.15,Z 389.977,A -85,B 0,C 180,E1 -11280.535,E2 -11280.535} C_VEL
LIN {X 0,Y 398.416,Z 377.026,A -85,B 0,C 180,E1 -11284.366,E2 -11284.366} C_VEL
LIN {X 0,Y 397.137,Z 371.016,A -85,B 0,C 180,E1 -11286.28,E2 -11286.28} C_VEL
LIN {X 0,Y 397.114,Z 371.018,A -85,B 0,C 180,E1 -11289.577,E2 -11289.577} C_VEL
LIN {X 0,Y 397.106,Z 371.019,A -85,B 0,C 180,E1 -11293.479,E2 -11293.479} C_VEL
LIN {X 0,Y 397.106,Z 371.022,A -85,B 0,C 180,E1 -11296.52,E2 -11296.52} C_VEL
LIN {X 0,Y 397.115,Z 371.017,A -85,B 0,C 180,E1 -11299.552,E2 -11299.552} C_VEL
LIN {X 0,Y 397.099,Z 371.02,A -85,B 0,C 180,E1 -11302.79,E2 -11302.79} C_VEL
LIN {X 0,Y 397.119,Z 371.02,A -85,B 0,C 180,E1 -11306.282,E2 -11306.282} C_VEL
LIN {X 0,Y 397.106,Z 371.022,A -85,B 0,C 180,E1 -11310.135,E2 -11310.135} C_VEL
LIN {X 0,Y 397.195,Z 371.007,A -85,B 0,C 180,E1 -11312.61,E2 -11312.61} C_VEL
LIN {X 0,Y 397.134,Z 371.017,A -85,B 0,C 180,E1 -11315.982,E2 -11315.982} C_VEL
LIN {X 0,Y 397.139,Z 371.017,A -85,B 0,C 180,E1 -11319.705,E2 -11319.705} C_VEL
LIN {X 0,Y 397.183,Z 371.007,A -85,B 0,C 180,E1 -11322.845,E2 -11322.845} C_VEL
LIN {X 0,Y 397.227,Z 371.003,A -85,B 0,C 180,E1 -11326.679,E2 -11326.679} C_VEL
LIN {X 0,Y 397.219,Z 371.008,A -85,B 0,C 180,E1 -11329.809,E2 -11329.809} C_VEL
LIN {X 0,Y 397.365,Z 370.985,A -85,B 0,C 180,E1 -11332.888,E2 -11332.888} C_VEL
LIN {X 0,Y 397.257,Z 371,A -85,B 0,C 180,E1 -11334.925,E2 -11334.925} C_VEL
LIN {X 0,Y 397.453,Z 370.978,A -85,B 0,C 180,E1 -11337.973,E2 -11337.973} C_VEL
LIN {X 0,Y 397.582,Z 370.961,A -85,B 0,C 180,E1 -11340,E2 -11340} C_VEL
LIN {X 0,Y 397.377,Z 370.986,A -85,B 0,C 180,E1 -11343.041,E2 -11343.041} C_VEL
LIN {X 0,Y 397.365,Z 370.989,A -85,B 0,C 180,E1 -11347.112,E2 -11347.112} C_VEL
LIN {X 0,Y 397.23,Z 371.003,A -85,B 0,C 180,E1 -11350.191,E2 -11350.191} C_VEL
LIN {X 0,Y 397.227,Z 371.007,A -85,B 0,C 180,E1 -11353.321,E2 -11353.321} C_VEL
LIN {X 0,Y 397.183,Z 371.013,A -85,B 0,C 180,E1 -11357.155,E2 -11357.155} C_VEL
LIN {X 0,Y 397.104,Z 371.021,A -85,B 0,C 180,E1 -11360.73,E2 -11360.73} C_VEL
LIN {X 0,Y 397.134,Z 371.015,A -85,B 0,C 180,E1 -11364.018,E2 -11364.018} C_VEL
LIN {X 0,Y 397.195,Z 371.009,A -85,B 0,C 180,E1 -11367.39,E2 -11367.39} C_VEL
LIN {X 0,Y 397.08,Z 371.025,A -85,B 0,C 180,E1 -11370.883,E2 -11370.883} C_VEL
LIN {X 0,Y 397.127,Z 371.017,A -85,B 0,C 180,E1 -11374.493,E2 -11374.493} C_VEL
LIN {X 0,Y 397.106,Z 371.018,A -85,B 0,C 180,E1 -11378.275,E2 -11378.275} C_VEL
LIN {X 0,Y 397.09,Z 371.023,A -85,B 0,C 180,E1 -11380.909,E2 -11380.909} C_VEL
LIN {X 0,Y 397.102,Z 371.019,A -85,B 0,C 180,E1 -11383.649,E2 -11383.649} C_VEL
LIN {X 0,Y 397.106,Z 371.021,A -85,B 0,C 180,E1 -11386.521,E2 -11386.521} C_VEL
LIN {X 0,Y 397.115,Z 371.02,A -85,B 0,C 180,E1 -11390.423,E2 -11390.423} C_VEL
LIN {X 0,Y 397.109,Z 371.021,A -85,B 0,C 180,E1 -11394.266,E2 -11394.266} C_VEL
LIN {X 0,Y 397.116,Z 371.021,A -85,B 0,C 180,E1 -11396.727,E2 -11396.727} C_VEL
LIN {X 0,Y 397.126,Z 371.019,A -85,B 0,C 180,E1 -11400.296,E2 -11400.296} C_VEL
LIN {X 0,Y 397.196,Z 371.01,A -85,B 0,C 180,E1 -11402.61,E2 -11402.61} C_VEL
LIN {X 0,Y 397.135,Z 371.018,A -85,B 0,C 180,E1 -11405.982,E2 -11405.982} C_VEL
LIN {X 0,Y 397.157,Z 371.012,A -85,B 0,C 180,E1 -11409.699,E2 -11409.699} C_VEL
LIN {X 0,Y 397.186,Z 371.009,A -85,B 0,C 180,E1 -11412.844,E2 -11412.844} C_VEL
LIN {X 0,Y 397.181,Z 371.01,A -85,B 0,C 180,E1 -11415.657,E2 -11415.657} C_VEL
LIN {X 0,Y 397.202,Z 371.007,A -85,B 0,C 180,E1 -11418.777,E2 -11418.777} C_VEL
LIN {X 0,Y 397.364,Z 370.991,A -85,B 0,C 180,E1 -11422.076,E2 -11422.076} C_VEL
LIN {X 0,Y 397.257,Z 371,A -85,B 0,C 180,E1 -11424.925,E2 -11424.925} C_VEL
LIN {X 0,Y 397.453,Z 370.978,A -85,B 0,C 180,E1 -11427.973,E2 -11427.973} C_VEL
LIN {X 0,Y 397.584,Z 370.962,A -85,B 0,C 180,E1 -11430,E2 -11430} C_VEL
LIN {X 0,Y 397.378,Z 370.983,A -85,B 0,C 180,E1 -11433.042,E2 -11433.042} C_VEL
LIN {X 0,Y 397.373,Z 370.987,A -85,B 0,C 180,E1 -11436.092,E2 -11436.092} C_VEL
LIN {X 0,Y 397.256,Z 371.001,A -85,B 0,C 180,E1 -11439.162,E2 -11439.162} C_VEL
LIN {X 0,Y 397.223,Z 371.005,A -85,B 0,C 180,E1 -11442.258,E2 -11442.258} C_VEL
LIN {X 0,Y 397.183,Z 371.011,A -85,B 0,C 180,E1 -11445.392,E2 -11445.392} C_VEL
LIN {X 0,Y 397.165,Z 371.011,A -85,B 0,C 180,E1 -11448.574,E2 -11448.574} C_VEL
LIN {X 0,Y 397.095,Z 371.023,A -85,B 0,C 180,E1 -11451.908,E2 -11451.908} C_VEL
LIN {X 0,Y 397.155,Z 371.017,A -85,B 0,C 180,E1 -11455.512,E2 -11455.512} C_VEL
LIN {X 0,Y 397.137,Z 371.014,A -85,B 0,C 180,E1 -11456.32,E2 -11456.32} C_VEL
LIN {X 0,Y 396.467,Z 371.101,A -85,B 0,C 180,E1 -11457.167,E2 -11457.167} C_VEL
LIN {X 0,Y 393.593,Z 371.456,A -85,B 0,C 180,E1 -11458.543,E2 -11458.543} C_VEL
LIN {X 0,Y 391.155,Z 371.762,A -85,B 0,C 180,E1 -11459.654,E2 -11459.654} C_VEL
LIN {X 0,Y 390.103,Z 371.891,A -85,B 0,C 180,E1 -11460.514,E2 -11460.514} C_VEL
LIN {X 0,Y 390.015,Z 371.901,A -85,B 0,C 180,E1 -11460.805,E2 -11460.805} C_VEL
LIN {X 0,Y 390.071,Z 371.895,A -85,B 0,C 180,E1 -11464.025,E2 -11464.025} C_VEL
LIN {X 0,Y 390.046,Z 371.9,A -85,B 0,C 180,E1 -11467.551,E2 -11467.551} C_VEL
LIN {X 0,Y 390.06,Z 371.898,A -85,B 0,C 180,E1 -11470.822,E2 -11470.822} C_VEL
LIN {X 0,Y 390.059,Z 371.897,A -85,B 0,C 180,E1 -11473.887,E2 -11473.887} C_VEL
LIN {X 0,Y 390.06,Z 371.897,A -85,B 0,C 180,E1 -11476.79,E2 -11476.79} C_VEL
LIN {X 0,Y 390.059,Z 371.898,A -85,B 0,C 180,E1 -11479.561,E2 -11479.561} C_VEL
LIN {X 0,Y 390.049,Z 371.898,A -85,B 0,C 180,E1 -11482.449,E2 -11482.449} C_VEL
LIN {X 0,Y 390.087,Z 371.892,A -85,B 0,C 180,E1 -11486.047,E2 -11486.047} C_VEL
LIN {X 0,Y 390.255,Z 371.952,A -85,B 0,C 180,E1 -11488.969,E2 -11488.969} C_VEL
LIN {X 0,Y 390.286,Z 375.368,A -85,B 0,C 180,E1 -11490.909,E2 -11490.909} C_VEL
LIN {X 0,Y 389.947,Z 381.633,A -85,B 0,C 180,E1 -11494.37,E2 -11494.37} C_VEL
LIN {X 0,Y 389.692,Z 387.812,A -85,B 0,C 180,E1 -11497.745,E2 -11497.745} C_VEL
LIN {X 0,Y 389.516,Z 393.997,A -85,B 0,C 180,E1 -11501.048,E2 -11501.048} C_VEL
LIN {X 0,Y 389.365,Z 400.139,A -85,B 0,C 180,E1 -11504.291,E2 -11504.291} C_VEL
LIN {X 0,Y 389.2,Z 407.392,A -85,B 0,C 180,E1 -11508.015,E2 -11508.015} C_VEL
LIN {X 0,Y 389.114,Z 409.517,A -85,B 0,C 180,E1 -11509.101,E2 -11509.101} C_VEL
LIN {X 0,Y 390.599,Z 420.712,A -85,B 0,C 180,E1 -11509.765,E2 -11509.765} C_VEL
LIN {X 0,Y 391.035,Z 426.262,A -85,B 0,C 180,E1 -11510.169,E2 -11510.169} C_VEL
LIN {X 0,Y 390.621,Z 436.481,A -85,B 0,C 180,E1 -11511.073,E2 -11511.073} C_VEL
LIN {X 0,Y 390.187,Z 445.872,A -85,B 0,C 180,E1 -11512.162,E2 -11512.162} C_VEL
LIN {X 0,Y 390.001,Z 453.282,A -85,B 0,C 180,E1 -11513.273,E2 -11513.273} C_VEL
LIN {X 0,Y 389.788,Z 460.025,A -85,B 0,C 180,E1 -11514.568,E2 -11514.568} C_VEL
LIN {X 0,Y 389.544,Z 465.159,A -85,B 0,C 180,E1 -11515.862,E2 -11515.862} C_VEL
LIN {X 0,Y 389.299,Z 468.319,A -85,B 0,C 180,E1 -11516.895,E2 -11516.895} C_VEL
LIN {X 0,Y 389.186,Z 470.7,A -85,B 0,C 180,E1 -11517.93,E2 -11517.93} C_VEL
LIN {X 0,Y 389.082,Z 472.37,A -85,B 0,C 180,E1 -11518.965,E2 -11518.965} C_VEL
LIN {X 0,Y 389.072,Z 473.354,A -85,B 0,C 180,E1 -11520,E2 -11520} C_VEL
LIN {X 0,Y 389.133,Z 473.668,A -85,B 0,C 180,E1 -11521.035,E2 -11521.035} C_VEL
LIN {X 0,Y 389.261,Z 473.317,A -85,B 0,C 180,E1 -11522.069,E2 -11522.069} C_VEL
LIN {X 0,Y 389.473,Z 472.305,A -85,B 0,C 180,E1 -11523.103,E2 -11523.103} C_VEL
LIN {X 0,Y 390.119,Z 469.482,A -85,B 0,C 180,E1 -11524.65,E2 -11524.65} C_VEL
LIN {X 0,Y 390.402,Z 466.724,A -85,B 0,C 180,E1 -11525.682,E2 -11525.682} C_VEL
LIN {X 0,Y 390.942,Z 462.104,A -85,B 0,C 180,E1 -11526.97,E2 -11526.97} C_VEL
LIN {X 0,Y 391.554,Z 456.025,A -85,B 0,C 180,E1 -11528.256,E2 -11528.256} C_VEL
LIN {X 0,Y 392.387,Z 448.102,A -85,B 0,C 180,E1 -11529.543,E2 -11529.543} C_VEL
LIN {X 0,Y 393.191,Z 439.511,A -85,B 0,C 180,E1 -11530.622,E2 -11530.622} C_VEL
LIN {X 0,Y 393.798,Z 431.137,A -85,B 0,C 180,E1 -11531.452,E2 -11531.452} C_VEL
LIN {X 0,Y 392.286,Z 422.211,A -85,B 0,C 180,E1 -11532.283,E2 -11532.283} C_VEL
LIN {X 0,Y 390.156,Z 413.58,A -85,B 0,C 180,E1 -11533.006,E2 -11533.006} C_VEL
LIN {X 0,Y 390.459,Z 407.357,A -85,B 0,C 180,E1 -11536.738,E2 -11536.738} C_VEL
LIN {X 0,Y 390.888,Z 402.184,A -85,B 0,C 180,E1 -11539.975,E2 -11539.975} C_VEL
LIN {X 0,Y 391.466,Z 396.549,A -85,B 0,C 180,E1 -11543.707,E2 -11543.707} C_VEL
LIN {X 0,Y 391.989,Z 392.416,A -85,B 0,C 180,E1 -11546.63,E2 -11546.63} C_VEL
LIN {X 0,Y 392.48,Z 389.432,A -85,B 0,C 180,E1 -11548.913,E2 -11548.913} C_VEL
LIN {X 0,Y 392.711,Z 386.696,A -85,B 0,C 180,E1 -11551.264,E2 -11551.264} C_VEL
LIN {X 0,Y 392.597,Z 384.304,A -85,B 0,C 180,E1 -11553.707,E2 -11553.707} C_VEL
LIN {X 0,Y 392.339,Z 382.321,A -85,B 0,C 180,E1 -11556.284,E2 -11556.284} C_VEL
LIN {X 0,Y 392.132,Z 380.94,A -85,B 0,C 180,E1 -11558.851,E2 -11558.851} C_VEL
LIN {X 0,Y 392.042,Z 380.214,A -85,B 0,C 180,E1 -11561.551,E2 -11561.551} C_VEL
LIN {X 0,Y 392.179,Z 380.409,A -85,B 0,C 180,E1 -11564.339,E2 -11564.339} C_VEL
LIN {X 0,Y 392.519,Z 381.677,A -85,B 0,C 180,E1 -11567.231,E2 -11567.231} C_VEL
LIN {X 0,Y 393.15,Z 384.243,A -85,B 0,C 180,E1 -11570.235,E2 -11570.235} C_VEL
LIN {X 0,Y 394.116,Z 388.328,A -85,B 0,C 180,E1 -11573.365,E2 -11573.365} C_VEL
LIN {X 0,Y 395.189,Z 392.732,A -85,B 0,C 180,E1 -11575.931,E2 -11575.931} C_VEL
LIN {X 0,Y 396.203,Z 397.872,A -85,B 0,C 180,E1 -11578.369,E2 -11578.369} C_VEL
LIN {X 0,Y 396.572,Z 401.02,A -85,B 0,C 180,E1 -11579.663,E2 -11579.663} C_VEL
LIN {X 0,Y 396.108,Z 404.285,A -85,B 0,C 180,E1 -11580.827,E2 -11580.827} C_VEL
LIN {X 0,Y 393.987,Z 414.553,A -85,B 0,C 180,E1 -11584.085,E2 -11584.085} C_VEL
LIN {X 0,Y 392.376,Z 425.644,A -85,B 0,C 180,E1 -11587.35,E2 -11587.35} C_VEL
LIN {X 0,Y 390.959,Z 439.453,A -85,B 0,C 180,E1 -11591.121,E2 -11591.121} C_VEL
LIN {X 0,Y 390.81,Z 441.182,A -85,B 0,C 180,E1 -11591.572,E2 -11591.572} C_VEL
LIN {X 0,Y 392.762,Z 453.445,A -85,B 0,C 180,E1 -11592.119,E2 -11592.119} C_VEL
LIN {X 0,Y 393.502,Z 464.416,A -85,B 0,C 180,E1 -11592.71,E2 -11592.71} C_VEL
LIN {X 0,Y 393.62,Z 473.348,A -85,B 0,C 180,E1 -11593.286,E2 -11593.286} C_VEL
LIN {X 0,Y 392.72,Z 484.811,A -85,B 0,C 180,E1 -11594.162,E2 -11594.162} C_VEL
LIN {X 0,Y 391.84,Z 495.456,A -85,B 0,C 180,E1 -11595.191,E2 -11595.191} C_VEL
LIN {X 0,Y 390.957,Z 506.143,A -85,B 0,C 180,E1 -11596.485,E2 -11596.485} C_VEL
LIN {X 0,Y 390.2,Z 514.868,A -85,B 0,C 180,E1 -11597.782,E2 -11597.782} C_VEL
LIN {X 0,Y 389.555,Z 523.353,A -85,B 0,C 180,E1 -11599.343,E2 -11599.343} C_VEL
LIN {X 0,Y 389.188,Z 530.202,A -85,B 0,C 180,E1 -11600.908,E2 -11600.908} C_VEL
LIN {X 0,Y 389.015,Z 536.449,A -85,B 0,C 180,E1 -11602.735,E2 -11602.735} C_VEL
LIN {X 0,Y 388.929,Z 540.501,A -85,B 0,C 180,E1 -11604.296,E2 -11604.296} C_VEL
LIN {X 0,Y 388.934,Z 543.469,A -85,B 0,C 180,E1 -11605.855,E2 -11605.855} C_VEL
LIN {X 0,Y 389.059,Z 544.891,A -85,B 0,C 180,E1 -11606.893,E2 -11606.893} C_VEL
LIN {X 0,Y 389.117,Z 545.885,A -85,B 0,C 180,E1 -11607.93,E2 -11607.93} C_VEL
LIN {X 0,Y 389.021,Z 546.389,A -85,B 0,C 180,E1 -11608.965,E2 -11608.965} C_VEL
LIN {X 0,Y 388.994,Z 546.482,A -85,B 0,C 180,E1 -11610,E2 -11610} C_VEL
LIN {X 0,Y 389.019,Z 546.167,A -85,B 0,C 180,E1 -11611.035,E2 -11611.035} C_VEL
LIN {X 0,Y 389.127,Z 545.384,A -85,B 0,C 180,E1 -11612.07,E2 -11612.07} C_VEL
LIN {X 0,Y 389.12,Z 544.154,A -85,B 0,C 180,E1 -11613.106,E2 -11613.106} C_VEL
LIN {X 0,Y 388.957,Z 541.423,A -85,B 0,C 180,E1 -11614.664,E2 -11614.664} C_VEL
LIN {X 0,Y 389.019,Z 537.596,A -85,B 0,C 180,E1 -11616.223,E2 -11616.223} C_VEL
LIN {X 0,Y 389.073,Z 532.535,A -85,B 0,C 180,E1 -11617.786,E2 -11617.786} C_VEL
LIN {X 0,Y 389.277,Z 526.031,A -85,B 0,C 180,E1 -11619.351,E2 -11619.351} C_VEL
LIN {X 0,Y 389.647,Z 517.841,A -85,B 0,C 180,E1 -11620.917,E2 -11620.917} C_VEL
LIN {X 0,Y 390.047,Z 509.387,A -85,B 0,C 180,E1 -11622.223,E2 -11622.223} C_VEL
LIN {X 0,Y 390.589,Z 501.207,A -85,B 0,C 180,E1 -11623.262,E2 -11623.262} C_VEL
LIN {X 0,Y 391.199,Z 491.53,A -85,B 0,C 180,E1 -11624.275,E2 -11624.275} C_VEL
LIN {X 0,Y 391.829,Z 480.39,A -85,B 0,C 180,E1 -11625.208,E2 -11625.208} C_VEL
LIN {X 0,Y 392.23,Z 468.335,A -85,B 0,C 180,E1 -11625.991,E2 -11625.991} C_VEL
LIN {X 0,Y 391.178,Z 455.414,A -85,B 0,C 180,E1 -11626.622,E2 -11626.622} C_VEL
LIN {X 0,Y 390.138,Z 442.716,A -85,B 0,C 180,E1 -11627.056,E2 -11627.056} C_VEL
LIN {X 0,Y 391.057,Z 429.54,A -85,B 0,C 180,E1 -11630.438,E2 -11630.438} C_VEL
LIN {X 0,Y 392.3,Z 415.928,A -85,B 0,C 180,E1 -11633.984,E2 -11633.984} C_VEL
LIN {X 0,Y 393.852,Z 402.115,A -85,B 0,C 180,E1 -11637.642,E2 -11637.642} C_VEL
LIN {X 0,Y 394.683,Z 395.196,A -85,B 0,C 180,E1 -11639.493,E2 -11639.493} C_VEL
LIN {X 0,Y 393.775,Z 389.401,A -85,B 0,C 180,E1 -11641.17,E2 -11641.17} C_VEL
LIN {X 0,Y 391.38,Z 377.941,A -85,B 0,C 180,E1 -11644.65,E2 -11644.65} C_VEL
LIN {X 0,Y 390.077,Z 371.895,A -85,B 0,C 180,E1 -11646.561,E2 -11646.561} C_VEL
LIN {X 0,Y 390.07,Z 371.895,A -85,B 0,C 180,E1 -11649.218,E2 -11649.218} C_VEL
LIN {X 0,Y 390.046,Z 371.901,A -85,B 0,C 180,E1 -11652.374,E2 -11652.374} C_VEL
LIN {X 0,Y 390.049,Z 371.898,A -85,B 0,C 180,E1 -11655.355,E2 -11655.355} C_VEL
LIN {X 0,Y 390.045,Z 371.901,A -85,B 0,C 180,E1 -11658.188,E2 -11658.188} C_VEL
LIN {X 0,Y 390.093,Z 371.891,A -85,B 0,C 180,E1 -11660.908,E2 -11660.908} C_VEL
LIN {X 0,Y 390.086,Z 371.893,A -85,B 0,C 180,E1 -11664.793,E2 -11664.793} C_VEL
LIN {X 0,Y 390.032,Z 371.902,A -85,B 0,C 180,E1 -11667.875,E2 -11667.875} C_VEL
LIN {X 0,Y 390.059,Z 371.895,A -85,B 0,C 180,E1 -11670.89,E2 -11670.89} C_VEL
LIN {X 0,Y 390.12,Z 371.891,A -85,B 0,C 180,E1 -11674.256,E2 -11674.256} C_VEL
LIN {X 0,Y 390.041,Z 371.901,A -85,B 0,C 180,E1 -11677.766,E2 -11677.766} C_VEL
LIN {X 0,Y 390.107,Z 371.89,A -85,B 0,C 180,E1 -11681.078,E2 -11681.078} C_VEL
LIN {X 0,Y 390.141,Z 371.887,A -85,B 0,C 180,E1 -11684.323,E2 -11684.323} C_VEL
LIN {X 0,Y 390.172,Z 371.885,A -85,B 0,C 180,E1 -11687.517,E2 -11687.517} C_VEL
LIN {X 0,Y 390.315,Z 371.869,A -85,B 0,C 180,E1 -11691.718,E2 -11691.718} C_VEL
LIN {X 0,Y 390.331,Z 371.865,A -85,B 0,C 180,E1 -11693.798,E2 -11693.798} C_VEL
LIN {X 0,Y 390.422,Z 371.854,A -85,B 0,C 180,E1 -11697.937,E2 -11697.937} C_VEL
LIN {X 0,Y 390.552,Z 371.837,A -85,B 0,C 180,E1 -11700,E2 -11700} C_VEL
LIN {X 0,Y 390.311,Z 371.866,A -85,B 0,C 180,E1 -11703.097,E2 -11703.097} C_VEL
LIN {X 0,Y 390.311,Z 371.864,A -85,B 0,C 180,E1 -11706.648,E2 -11706.648} C_VEL
LIN {X 0,Y 390.211,Z 371.88,A -85,B 0,C 180,E1 -11709.329,E2 -11709.329} C_VEL
LIN {X 0,Y 390.179,Z 371.881,A -85,B 0,C 180,E1 -11712.483,E2 -11712.483} C_VEL
LIN {X 0,Y 390.141,Z 371.887,A -85,B 0,C 180,E1 -11715.677,E2 -11715.677} C_VEL
LIN {X 0,Y 390.107,Z 371.894,A -85,B 0,C 180,E1 -11718.922,E2 -11718.922} C_VEL
LIN {X 0,Y 390.041,Z 371.898,A -85,B 0,C 180,E1 -11722.234,E2 -11722.234} C_VEL
LIN {X 0,Y 390.12,Z 371.888,A -85,B 0,C 180,E1 -11725.744,E2 -11725.744} C_VEL
LIN {X 0,Y 390.06,Z 371.899,A -85,B 0,C 180,E1 -11729.11,E2 -11729.11} C_VEL
LIN {X 0,Y 390.044,Z 371.901,A -85,B 0,C 180,E1 -11732.722,E2 -11732.722} C_VEL
LIN {X 0,Y 390.058,Z 371.895,A -85,B 0,C 180,E1 -11735.826,E2 -11735.826} C_VEL
LIN {X 0,Y 390.072,Z 371.896,A -85,B 0,C 180,E1 -11739.219,E2 -11739.219} C_VEL
LIN {X 0,Y 390.043,Z 371.901,A -85,B 0,C 180,E1 -11742.374,E2 -11742.374} C_VEL
LIN {X 0,Y 390.048,Z 371.898,A -85,B 0,C 180,E1 -11745.355,E2 -11745.355} C_VEL
LIN {X 0,Y 390.034,Z 371.9,A -85,B 0,C 180,E1 -11748.187,E2 -11748.187} C_VEL
LIN {X 0,Y 390.092,Z 371.894,A -85,B 0,C 180,E1 -11750.908,E2 -11750.908} C_VEL
LIN {X 0,Y 390.086,Z 371.896,A -85,B 0,C 180,E1 -11754.793,E2 -11754.793} C_VEL
LIN {X 0,Y 390.026,Z 371.904,A -85,B 0,C 180,E1 -11758.496,E2 -11758.496} C_VEL
LIN {X 0,Y 390.119,Z 371.891,A -85,B 0,C 180,E1 -11762.07,E2 -11762.07} C_VEL
LIN {X 0,Y 390.082,Z 371.893,A -85,B 0,C 180,E1 -11765.52,E2 -11765.52} C_VEL
LIN {X 0,Y 390.074,Z 371.895,A -85,B 0,C 180,E1 -11768.879,E2 -11768.879} C_VEL
LIN {X 0,Y 390.134,Z 371.891,A -85,B 0,C 180,E1 -11772.167,E2 -11772.167} C_VEL
LIN {X 0,Y 390.149,Z 371.885,A -85,B 0,C 180,E1 -11775.393,E2 -11775.393} C_VEL
LIN {X 0,Y 390.151,Z 371.887,A -85,B 0,C 180,E1 -11778.571,E2 -11778.571} C_VEL
LIN {X 0,Y 390.31,Z 371.869,A -85,B 0,C 180,E1 -11782.032,E2 -11782.032} C_VEL
LIN {X 0,Y 390.228,Z 371.875,A -85,B 0,C 180,E1 -11784.834,E2 -11784.834} C_VEL
LIN {X 0,Y 390.421,Z 371.854,A -85,B 0,C 180,E1 -11787.937,E2 -11787.937} C_VEL
LIN {X 0,Y 390.553,Z 371.838,A -85,B 0,C 180,E1 -11790,E2 -11790} C_VEL
LIN {X 0,Y 390.313,Z 371.863,A -85,B 0,C 180,E1 -11793.097,E2 -11793.097} C_VEL
LIN {X 0,Y 390.327,Z 371.865,A -85,B 0,C 180,E1 -11796.202,E2 -11796.202} C_VEL
LIN {X 0,Y 390.208,Z 371.879,A -85,B 0,C 180,E1 -11799.329,E2 -11799.329} C_VEL
LIN {X 0,Y 390.174,Z 371.881,A -85,B 0,C 180,E1 -11802.483,E2 -11802.483} C_VEL
LIN {X 0,Y 390.143,Z 371.89,A -85,B 0,C 180,E1 -11805.677,E2 -11805.677} C_VEL
LIN {X 0,Y 390.109,Z 371.89,A -85,B 0,C 180,E1 -11808.922,E2 -11808.922} C_VEL
LIN {X 0,Y 390.042,Z 371.899,A -85,B 0,C 180,E1 -11812.234,E2 -11812.234} C_VEL
LIN {X 0,Y 390.122,Z 371.891,A -85,B 0,C 180,E1 -11815.743,E2 -11815.743} C_VEL
LIN {X 0,Y 390.061,Z 371.898,A -85,B 0,C 180,E1 -11819.11,E2 -11819.11} C_VEL
LIN {X 0,Y 390.015,Z 371.901,A -85,B 0,C 180,E1 -11820.805,E2 -11820.805} C_VEL
LIN {X 0,Y 389.341,Z 371.989,A -85,B 0,C 180,E1 -11821.667,E2 -11821.667} C_VEL
LIN {X 0,Y 386.494,Z 372.342,A -85,B 0,C 180,E1 -11823.069,E2 -11823.069} C_VEL
LIN {X 0,Y 384.096,Z 372.638,A -85,B 0,C 180,E1 -11824.202,E2 -11824.202} C_VEL
LIN {X 0,Y 383.078,Z 372.767,A -85,B 0,C 180,E1 -11825.077,E2 -11825.077} C_VEL
LIN {X 0,Y 383.001,Z 372.772,A -85,B 0,C 180,E1 -11825.374,E2 -11825.374} C_VEL
LIN {X 0,Y 383.007,Z 372.774,A -85,B 0,C 180,E1 -11828.601,E2 -11828.601} C_VEL
LIN {X 0,Y 382.988,Z 372.78,A -85,B 0,C 180,E1 -11831.347,E2 -11831.347} C_VEL
LIN {X 0,Y 383,Z 372.775,A -85,B 0,C 180,E1 -11834.304,E2 -11834.304} C_VEL
LIN {X 0,Y 383.013,Z 372.778,A -85,B 0,C 180,E1 -11837.24,E2 -11837.24} C_VEL
LIN {X 0,Y 383.019,Z 372.773,A -85,B 0,C 180,E1 -11840.413,E2 -11840.413} C_VEL
LIN {X 0,Y 383.03,Z 372.772,A -85,B 0,C 180,E1 -11844.045,E2 -11844.045} C_VEL
LIN {X 0,Y 383.069,Z 372.768,A -85,B 0,C 180,E1 -11847.856,E2 -11847.856} C_VEL
LIN {X 0,Y 383.21,Z 372.904,A -85,B 0,C 180,E1 -11848.948,E2 -11848.948} C_VEL
LIN {X 0,Y 383.158,Z 377.393,A -85,B 0,C 180,E1 -11851.517,E2 -11851.517} C_VEL
LIN {X 0,Y 382.843,Z 383.646,A -85,B 0,C 180,E1 -11855.025,E2 -11855.025} C_VEL
LIN {X 0,Y 382.594,Z 389.896,A -85,B 0,C 180,E1 -11858.445,E2 -11858.445} C_VEL
LIN {X 0,Y 382.442,Z 395.102,A -85,B 0,C 180,E1 -11861.241,E2 -11861.241} C_VEL
LIN {X 0,Y 382.274,Z 401.309,A -85,B 0,C 180,E1 -11864.539,E2 -11864.539} C_VEL
LIN {X 0,Y 382.124,Z 408.581,A -85,B 0,C 180,E1 -11868.328,E2 -11868.328} C_VEL
LIN {X 0,Y 382.067,Z 409.82,A -85,B 0,C 180,E1 -11868.964,E2 -11868.964} C_VEL
LIN {X 0,Y 383.542,Z 421.164,A -85,B 0,C 180,E1 -11869.642,E2 -11869.642} C_VEL
LIN {X 0,Y 383.969,Z 427.537,A -85,B 0,C 180,E1 -11870.119,E2 -11870.119} C_VEL
LIN {X 0,Y 383.547,Z 437.577,A -85,B 0,C 180,E1 -11871.04,E2 -11871.04} C_VEL
LIN {X 0,Y 383.124,Z 446.685,A -85,B 0,C 180,E1 -11872.128,E2 -11872.128} C_VEL
LIN {X 0,Y 382.909,Z 454.92,A -85,B 0,C 180,E1 -11873.413,E2 -11873.413} C_VEL
LIN {X 0,Y 382.664,Z 461.44,A -85,B 0,C 180,E1 -11874.731,E2 -11874.731} C_VEL
LIN {X 0,Y 382.497,Z 465.527,A -85,B 0,C 180,E1 -11875.785,E2 -11875.785} C_VEL
LIN {X 0,Y 382.196,Z 470.077,A -85,B 0,C 180,E1 -11877.365,E2 -11877.365} C_VEL
LIN {X 0,Y 382.03,Z 472.955,A -85,B 0,C 180,E1 -11878.946,E2 -11878.946} C_VEL
LIN {X 0,Y 382.016,Z 474.015,A -85,B 0,C 180,E1 -11880,E2 -11880} C_VEL
LIN {X 0,Y 382.077,Z 474.406,A -85,B 0,C 180,E1 -11881.054,E2 -11881.054} C_VEL
LIN {X 0,Y 382.214,Z 474.135,A -85,B 0,C 180,E1 -11882.108,E2 -11882.108} C_VEL
LIN {X 0,Y 382.441,Z 473.202,A -85,B 0,C 180,E1 -11883.16,E2 -11883.16} C_VEL
LIN {X 0,Y 383.113,Z 470.5,A -85,B 0,C 180,E1 -11884.735,E2 -11884.735} C_VEL
LIN {X 0,Y 383.613,Z 466.212,A -85,B 0,C 180,E1 -11886.311,E2 -11886.311} C_VEL
LIN {X 0,Y 384.226,Z 461.236,A -85,B 0,C 180,E1 -11887.621,E2 -11887.621} C_VEL
LIN {X 0,Y 385.001,Z 454.717,A -85,B 0,C 180,E1 -11888.926,E2 -11888.926} C_VEL
LIN {X 0,Y 385.893,Z 446.469,A -85,B 0,C 180,E1 -11890.196,E2 -11890.196} C_VEL
LIN {X 0,Y 386.722,Z 437.725,A -85,B 0,C 180,E1 -11891.239,E2 -11891.239} C_VEL
LIN {X 0,Y 387.122,Z 432.186,A -85,B 0,C 180,E1 -11891.785,E2 -11891.785} C_VEL
LIN {X 0,Y 385.403,Z 422.601,A -85,B 0,C 180,E1 -11892.73,E2 -11892.73} C_VEL
LIN {X 0,Y 383.241,Z 414.077,A -85,B 0,C 180,E1 -11893.48,E2 -11893.48} C_VEL
LIN {X 0,Y 383.671,Z 407.195,A -85,B 0,C 180,E1 -11897.725,E2 -11897.725} C_VEL
LIN {X 0,Y 384.146,Z 401.498,A -85,B 0,C 180,E1 -11901.463,E2 -11901.463} C_VEL
LIN {X 0,Y 384.762,Z 396.671,A -85,B 0,C 180,E1 -11904.842,E2 -11904.842} C_VEL
LIN {X 0,Y 385.488,Z 392.105,A -85,B 0,C 180,E1 -11908.295,E2 -11908.295} C_VEL
LIN {X 0,Y 385.913,Z 388.829,A -85,B 0,C 180,E1 -11911.136,E2 -11911.136} C_VEL
LIN {X 0,Y 385.878,Z 386.932,A -85,B 0,C 180,E1 -11913.12,E2 -11913.12} C_VEL
LIN {X 0,Y 385.645,Z 384.974,A -85,B 0,C 180,E1 -11915.674,E2 -11915.674} C_VEL
LIN {X 0,Y 385.476,Z 383.496,A -85,B 0,C 180,E1 -11918.374,E2 -11918.374} C_VEL
LIN {X 0,Y 385.393,Z 382.759,A -85,B 0,C 180,E1 -11921.033,E2 -11921.033} C_VEL
LIN {X 0,Y 385.484,Z 382.818,A -85,B 0,C 180,E1 -11923.852,E2 -11923.852} C_VEL
LIN {X 0,Y 385.807,Z 383.991,A -85,B 0,C 180,E1 -11926.774,E2 -11926.774} C_VEL
LIN {X 0,Y 386.414,Z 386.375,A -85,B 0,C 180,E1 -11929.808,E2 -11929.808} C_VEL
LIN {X 0,Y 386.968,Z 388.736,A -85,B 0,C 180,E1 -11931.866,E2 -11931.866} C_VEL
LIN {X 0,Y 387.976,Z 392.798,A -85,B 0,C 180,E1 -11934.603,E2 -11934.603} C_VEL
LIN {X 0,Y 389.05,Z 397.608,A -85,B 0,C 180,E1 -11937.184,E2 -11937.184} C_VEL
LIN {X 0,Y 389.718,Z 401.812,A -85,B 0,C 180,E1 -11939.072,E2 -11939.072} C_VEL
LIN {X 0,Y 389.5,Z 405.24,A -85,B 0,C 180,E1 -11940.393,E2 -11940.393} C_VEL
LIN {X 0,Y 387.008,Z 416.722,A -85,B 0,C 180,E1 -11944.161,E2 -11944.161} C_VEL
LIN {X 0,Y 385.328,Z 427.801,A -85,B 0,C 180,E1 -11947.479,E2 -11947.479} C_VEL
LIN {X 0,Y 383.942,Z 440.7,A -85,B 0,C 180,E1 -11951.088,E2 -11951.088} C_VEL
LIN {X 0,Y 386.102,Z 454.207,A -85,B 0,C 180,E1 -11951.757,E2 -11951.757} C_VEL
LIN {X 0,Y 386.816,Z 465.531,A -85,B 0,C 180,E1 -11952.407,E2 -11952.407} C_VEL
LIN {X 0,Y 386.77,Z 475.53,A -85,B 0,C 180,E1 -11953.098,E2 -11953.098} C_VEL
LIN {X 0,Y 385.667,Z 487.886,A -85,B 0,C 180,E1 -11954.136,E2 -11954.136} C_VEL
LIN {X 0,Y 384.639,Z 499.084,A -85,B 0,C 180,E1 -11955.333,E2 -11955.333} C_VEL
LIN {X 0,Y 383.668,Z 509.661,A -85,B 0,C 180,E1 -11956.763,E2 -11956.763} C_VEL
LIN {X 0,Y 383.013,Z 517.639,A -85,B 0,C 180,E1 -11958.087,E2 -11958.087} C_VEL
LIN {X 0,Y 382.335,Z 525.429,A -85,B 0,C 180,E1 -11959.675,E2 -11959.675} C_VEL
LIN {X 0,Y 382.02,Z 532.645,A -85,B 0,C 180,E1 -11961.536,E2 -11961.536} C_VEL
LIN {X 0,Y 381.903,Z 537.557,A -85,B 0,C 180,E1 -11963.183,E2 -11963.183} C_VEL
LIN {X 0,Y 381.871,Z 541.05,A -85,B 0,C 180,E1 -11964.72,E2 -11964.72} C_VEL
LIN {X 0,Y 381.849,Z 542.861,A -85,B 0,C 180,E1 -11965.778,E2 -11965.778} C_VEL
LIN {X 0,Y 381.99,Z 544.263,A -85,B 0,C 180,E1 -11966.836,E2 -11966.836} C_VEL
LIN {X 0,Y 382.05,Z 545.214,A -85,B 0,C 180,E1 -11967.891,E2 -11967.891} C_VEL
LIN {X 0,Y 381.972,Z 545.691,A -85,B 0,C 180,E1 -11968.946,E2 -11968.946} C_VEL
LIN {X 0,Y 381.942,Z 545.761,A -85,B 0,C 180,E1 -11970,E2 -11970} C_VEL
LIN {X 0,Y 381.97,Z 545.406,A -85,B 0,C 180,E1 -11971.054,E2 -11971.054} C_VEL
LIN {X 0,Y 382.079,Z 544.585,A -85,B 0,C 180,E1 -11972.108,E2 -11972.108} C_VEL
LIN {X 0,Y 382.05,Z 543.326,A -85,B 0,C 180,E1 -11973.163,E2 -11973.163} C_VEL
LIN {X 0,Y 381.891,Z 540.533,A -85,B 0,C 180,E1 -11974.75,E2 -11974.75} C_VEL
LIN {X 0,Y 381.986,Z 536.101,A -85,B 0,C 180,E1 -11976.522,E2 -11976.522} C_VEL
LIN {X 0,Y 382.06,Z 530.456,A -85,B 0,C 180,E1 -11978.196,E2 -11978.196} C_VEL
LIN {X 0,Y 382.259,Z 523.603,A -85,B 0,C 180,E1 -11979.791,E2 -11979.791} C_VEL
LIN {X 0,Y 382.616,Z 516.542,A -85,B 0,C 180,E1 -11981.12,E2 -11981.12} C_VEL
LIN {X 0,Y 383.055,Z 507.881,A -85,B 0,C 180,E1 -11982.449,E2 -11982.449} C_VEL
LIN {X 0,Y 383.504,Z 500.678,A -85,B 0,C 180,E1 -11983.376,E2 -11983.376} C_VEL
LIN {X 0,Y 384.26,Z 489.607,A -85,B 0,C 180,E1 -11984.538,E2 -11984.538} C_VEL
LIN {X 0,Y 384.898,Z 478.155,A -85,B 0,C 180,E1 -11985.488,E2 -11985.488} C_VEL
LIN {X 0,Y 385.208,Z 468.979,A -85,B 0,C 180,E1 -11986.087,E2 -11986.087} C_VEL
LIN {X 0,Y 384.185,Z 456.179,A -85,B 0,C 180,E1 -11986.745,E2 -11986.745} C_VEL
LIN {X 0,Y 383.095,Z 442.421,A -85,B 0,C 180,E1 -11987.239,E2 -11987.239} C_VEL
LIN {X 0,Y 384.063,Z 429.218,A -85,B 0,C 180,E1 -11990.723,E2 -11990.723} C_VEL
LIN {X 0,Y 385.346,Z 416.066,A -85,B 0,C 180,E1 -11994.229,E2 -11994.229} C_VEL
LIN {X 0,Y 386.925,Z 402.5,A -85,B 0,C 180,E1 -11997.886,E2 -11997.886} C_VEL
LIN {X 0,Y 387.663,Z 396.581,A -85,B 0,C 180,E1 -11999.518,E2 -11999.518} C_VEL
LIN {X 0,Y 387.323,Z 393.095,A -85,B 0,C 180,E1 -12000.535,E2 -12000.535} C_VEL
LIN {X 0,Y 384.599,Z 380.177,A -85,B 0,C 180,E1 -12004.505,E2 -12004.505} C_VEL
LIN {X 0,Y 383.037,Z 372.772,A -85,B 0,C 180,E1 -12006.911,E2 -12006.911} C_VEL
LIN {X 0,Y 383.009,Z 372.777,A -85,B 0,C 180,E1 -12009.958,E2 -12009.958} C_VEL
LIN {X 0,Y 383.006,Z 372.776,A -85,B 0,C 180,E1 -12012.778,E2 -12012.778} C_VEL
LIN {X 0,Y 383.002,Z 372.777,A -85,B 0,C 180,E1 -12015.79,E2 -12015.79} C_VEL
LIN {X 0,Y 383.003,Z 372.775,A -85,B 0,C 180,E1 -12018.793,E2 -12018.793} C_VEL
LIN {X 0,Y 383.003,Z 372.779,A -85,B 0,C 180,E1 -12022.096,E2 -12022.096} C_VEL
LIN {X 0,Y 383.019,Z 372.773,A -85,B 0,C 180,E1 -12025.332,E2 -12025.332} C_VEL
LIN {X 0,Y 382.984,Z 372.777,A -85,B 0,C 180,E1 -12029.081,E2 -12029.081} C_VEL
LIN {X 0,Y 383.057,Z 372.768,A -85,B 0,C 180,E1 -12032.698,E2 -12032.698} C_VEL
LIN {X 0,Y 383.034,Z 372.774,A -85,B 0,C 180,E1 -12036.193,E2 -12036.193} C_VEL
LIN {X 0,Y 383.056,Z 372.771,A -85,B 0,C 180,E1 -12039.598,E2 -12039.598} C_VEL
LIN {X 0,Y 383.106,Z 372.761,A -85,B 0,C 180,E1 -12042.931,E2 -12042.931} C_VEL
LIN {X 0,Y 383.126,Z 372.76,A -85,B 0,C 180,E1 -12046.464,E2 -12046.464} C_VEL
LIN {X 0,Y 383.153,Z 372.756,A -85,B 0,C 180,E1 -12050.498,E2 -12050.498} C_VEL
LIN {X 0,Y 383.274,Z 372.74,A -85,B 0,C 180,E1 -12052.625,E2 -12052.625} C_VEL
LIN {X 0,Y 383.201,Z 372.75,A -85,B 0,C 180,E1 -12054.739,E2 -12054.739} C_VEL
LIN {X 0,Y 383.389,Z 372.73,A -85,B 0,C 180,E1 -12057.899,E2 -12057.899} C_VEL
LIN {X 0,Y 383.521,Z 372.712,A -85,B 0,C 180,E1 -12060,E2 -12060} C_VEL
LIN {X 0,Y 383.248,Z 372.746,A -85,B 0,C 180,E1 -12063.154,E2 -12063.154} C_VEL
LIN {X 0,Y 383.27,Z 372.741,A -85,B 0,C 180,E1 -12066.643,E2 -12066.643} C_VEL
LIN {X 0,Y 383.262,Z 372.743,A -85,B 0,C 180,E1 -12068.436,E2 -12068.436} C_VEL
LIN {X 0,Y 383.109,Z 372.765,A -85,B 0,C 180,E1 -12071.642,E2 -12071.642} C_VEL
LIN {X 0,Y 383.113,Z 372.763,A -85,B 0,C 180,E1 -12074.882,E2 -12074.882} C_VEL
LIN {X 0,Y 383.064,Z 372.767,A -85,B 0,C 180,E1 -12078.174,E2 -12078.174} C_VEL
LIN {X 0,Y 382.994,Z 372.779,A -85,B 0,C 180,E1 -12081.531,E2 -12081.531} C_VEL
LIN {X 0,Y 383.053,Z 372.772,A -85,B 0,C 180,E1 -12084.96,E2 -12084.96} C_VEL
LIN {X 0,Y 383.041,Z 372.771,A -85,B 0,C 180,E1 -12088.493,E2 -12088.493} C_VEL
LIN {X 0,Y 383.01,Z 372.774,A -85,B 0,C 180,E1 -12092.15,E2 -12092.15} C_VEL
LIN {X 0,Y 383.019,Z 372.775,A -85,B 0,C 180,E1 -12094.668,E2 -12094.668} C_VEL
LIN {X 0,Y 383.002,Z 372.774,A -85,B 0,C 180,E1 -12097.904,E2 -12097.904} C_VEL
LIN {X 0,Y 382.985,Z 372.779,A -85,B 0,C 180,E1 -12101.348,E2 -12101.348} C_VEL
LIN {X 0,Y 382.998,Z 372.778,A -85,B 0,C 180,E1 -12104.304,E2 -12104.304} C_VEL
LIN {X 0,Y 383.011,Z 372.774,A -85,B 0,C 180,E1 -12107.24,E2 -12107.24} C_VEL
LIN {X 0,Y 383.017,Z 372.776,A -85,B 0,C 180,E1 -12110.414,E2 -12110.414} C_VEL
LIN {X 0,Y 383.026,Z 372.773,A -85,B 0,C 180,E1 -12114.045,E2 -12114.045} C_VEL
LIN {X 0,Y 382.988,Z 372.776,A -85,B 0,C 180,E1 -12117.578,E2 -12117.578} C_VEL
LIN {X 0,Y 382.994,Z 372.779,A -85,B 0,C 180,E1 -12120.3,E2 -12120.3} C_VEL
LIN {X 0,Y 383.082,Z 372.767,A -85,B 0,C 180,E1 -12124.021,E2 -12124.021} C_VEL
LIN {X 0,Y 383.015,Z 372.773,A -85,B 0,C 180,E1 -12127.336,E2 -12127.336} C_VEL
LIN {X 0,Y 383.075,Z 372.767,A -85,B 0,C 180,E1 -12130.717,E2 -12130.717} C_VEL
LIN {X 0,Y 383.088,Z 372.768,A -85,B 0,C 180,E1 -12134.027,E2 -12134.027} C_VEL
LIN {X 0,Y 383.139,Z 372.758,A -85,B 0,C 180,E1 -12137.284,E2 -12137.284} C_VEL
LIN {X 0,Y 383.157,Z 372.757,A -85,B 0,C 180,E1 -12140.498,E2 -12140.498} C_VEL
LIN {X 0,Y 383.283,Z 372.742,A -85,B 0,C 180,E1 -12143.684,E2 -12143.684} C_VEL
LIN {X 0,Y 383.389,Z 372.73,A -85,B 0,C 180,E1 -12147.899,E2 -12147.899} C_VEL
LIN {X 0,Y 383.523,Z 372.714,A -85,B 0,C 180,E1 -12150,E2 -12150} C_VEL
LIN {X 0,Y 383.25,Z 372.743,A -85,B 0,C 180,E1 -12153.154,E2 -12153.154} C_VEL
LIN {X 0,Y 383.283,Z 372.742,A -85,B 0,C 180,E1 -12156.317,E2 -12156.317} C_VEL
LIN {X 0,Y 383.155,Z 372.759,A -85,B 0,C 180,E1 -12159.502,E2 -12159.502} C_VEL
LIN {X 0,Y 383.128,Z 372.762,A -85,B 0,C 180,E1 -12163.536,E2 -12163.536} C_VEL
LIN {X 0,Y 383.098,Z 372.767,A -85,B 0,C 180,E1 -12167.455,E2 -12167.455} C_VEL
LIN {X 0,Y 383.032,Z 372.771,A -85,B 0,C 180,E1 -12170.647,E2 -12170.647} C_VEL
LIN {X 0,Y 383.036,Z 372.774,A -85,B 0,C 180,E1 -12173.807,E2 -12173.807} C_VEL
LIN {X 0,Y 383.083,Z 372.766,A -85,B 0,C 180,E1 -12176.123,E2 -12176.123} C_VEL
LIN {X 0,Y 382.995,Z 372.779,A -85,B 0,C 180,E1 -12179.7,E2 -12179.7} C_VEL
LIN {X 0,Y 383.006,Z 372.778,A -85,B 0,C 180,E1 -12183.401,E2 -12183.401} C_VEL
LIN {X 0,Y 383.001,Z 372.772,A -85,B 0,C 180,E1 -12185.374,E2 -12185.374} C_VEL
LIN {X 0,Y 382.364,Z 372.854,A -85,B 0,C 180,E1 -12186.252,E2 -12186.252} C_VEL
LIN {X 0,Y 379.568,Z 373.206,A -85,B 0,C 180,E1 -12187.68,E2 -12187.68} C_VEL
LIN {X 0,Y 377.163,Z 373.506,A -85,B 0,C 180,E1 -12188.834,E2 -12188.834} C_VEL
LIN {X 0,Y 376.093,Z 373.638,A -85,B 0,C 180,E1 -12189.726,E2 -12189.726} C_VEL
LIN {X 0,Y 375.986,Z 373.65,A -85,B 0,C 180,E1 -12190.028,E2 -12190.028} C_VEL
LIN {X 0,Y 375.934,Z 373.657,A -85,B 0,C 180,E1 -12193.766,E2 -12193.766} C_VEL
LIN {X 0,Y 375.936,Z 373.656,A -85,B 0,C 180,E1 -12196.811,E2 -12196.811} C_VEL
LIN {X 0,Y 375.967,Z 373.652,A -85,B 0,C 180,E1 -12200.538,E2 -12200.538} C_VEL
LIN {X 0,Y 375.968,Z 373.654,A -85,B 0,C 180,E1 -12203.495,E2 -12203.495} C_VEL
LIN {X 0,Y 376.009,Z 373.649,A -85,B 0,C 180,E1 -12207.257,E2 -12207.257} C_VEL
LIN {X 0,Y 376.186,Z 373.803,A -85,B 0,C 180,E1 -12208.895,E2 -12208.895} C_VEL
LIN {X 0,Y 376.131,Z 378.164,A -85,B 0,C 180,E1 -12211.426,E2 -12211.426} C_VEL
LIN {X 0,Y 375.794,Z 384.712,A -85,B 0,C 180,E1 -12215.115,E2 -12215.115} C_VEL
LIN {X 0,Y 375.552,Z 390.985,A -85,B 0,C 180,E1 -12218.597,E2 -12218.597} C_VEL
LIN {X 0,Y 375.33,Z 397.225,A -85,B 0,C 180,E1 -12222.003,E2 -12222.003} C_VEL
LIN {X 0,Y 375.192,Z 402.446,A -85,B 0,C 180,E1 -12224.797,E2 -12224.797} C_VEL
LIN {X 0,Y 375.06,Z 408.705,A -85,B 0,C 180,E1 -12228.105,E2 -12228.105} C_VEL
LIN {X 0,Y 375.017,Z 410.21,A -85,B 0,C 180,E1 -12228.823,E2 -12228.823} C_VEL
LIN {X 0,Y 376.368,Z 420.602,A -85,B 0,C 180,E1 -12229.442,E2 -12229.442} C_VEL
LIN {X 0,Y 376.958,Z 427.15,A -85,B 0,C 180,E1 -12229.934,E2 -12229.934} C_VEL
LIN {X 0,Y 376.514,Z 437.386,A -85,B 0,C 180,E1 -12230.871,E2 -12230.871} C_VEL
LIN {X 0,Y 376.077,Z 446.659,A -85,B 0,C 180,E1 -12231.981,E2 -12231.981} C_VEL
LIN {X 0,Y 375.865,Z 455.034,A -85,B 0,C 180,E1 -12233.289,E2 -12233.289} C_VEL
LIN {X 0,Y 375.595,Z 461.668,A -85,B 0,C 180,E1 -12234.632,E2 -12234.632} C_VEL
LIN {X 0,Y 375.434,Z 465.828,A -85,B 0,C 180,E1 -12235.706,E2 -12235.706} C_VEL
LIN {X 0,Y 375.117,Z 470.513,A -85,B 0,C 180,E1 -12237.315,E2 -12237.315} C_VEL
LIN {X 0,Y 374.978,Z 473.521,A -85,B 0,C 180,E1 -12238.926,E2 -12238.926} C_VEL
LIN {X 0,Y 374.961,Z 474.666,A -85,B 0,C 180,E1 -12240,E2 -12240} C_VEL
LIN {X 0,Y 375.024,Z 475.142,A -85,B 0,C 180,E1 -12241.074,E2 -12241.074} C_VEL
LIN {X 0,Y 375.167,Z 474.953,A -85,B 0,C 180,E1 -12242.147,E2 -12242.147} C_VEL
LIN {X 0,Y 375.411,Z 474.107,A -85,B 0,C 180,E1 -12243.22,E2 -12243.22} C_VEL
LIN {X 0,Y 376.11,Z 471.561,A -85,B 0,C 180,E1 -12244.824,E2 -12244.824} C_VEL
LIN {X 0,Y 376.663,Z 467.446,A -85,B 0,C 180,E1 -12246.428,E2 -12246.428} C_VEL
LIN {X 0,Y 377.468,Z 461.491,A -85,B 0,C 180,E1 -12248.027,E2 -12248.027} C_VEL
LIN {X 0,Y 378.327,Z 454.822,A -85,B 0,C 180,E1 -12249.355,E2 -12249.355} C_VEL
LIN {X 0,Y 379.319,Z 446.234,A -85,B 0,C 180,E1 -12250.677,E2 -12250.677} C_VEL
LIN {X 0,Y 380.248,Z 437.396,A -85,B 0,C 180,E1 -12251.731,E2 -12251.731} C_VEL
LIN {X 0,Y 380.33,Z 432.219,A -85,B 0,C 180,E1 -12252.269,E2 -12252.269} C_VEL
LIN {X 0,Y 378.572,Z 423.033,A -85,B 0,C 180,E1 -12253.201,E2 -12253.201} C_VEL
LIN {X 0,Y 376.279,Z 414.62,A -85,B 0,C 180,E1 -12253.991,E2 -12253.991} C_VEL
LIN {X 0,Y 376.734,Z 408.399,A -85,B 0,C 180,E1 -12257.934,E2 -12257.934} C_VEL
LIN {X 0,Y 377.214,Z 403.35,A -85,B 0,C 180,E1 -12261.319,E2 -12261.319} C_VEL
LIN {X 0,Y 377.775,Z 399.199,A -85,B 0,C 180,E1 -12264.275,E2 -12264.275} C_VEL
LIN {X 0,Y 378.49,Z 394.818,A -85,B 0,C 180,E1 -12267.659,E2 -12267.659} C_VEL
LIN {X 0,Y 378.959,Z 392.035,A -85,B 0,C 180,E1 -12270.048,E2 -12270.048} C_VEL
LIN {X 0,Y 379.098,Z 389.583,A -85,B 0,C 180,E1 -12272.522,E2 -12272.522} C_VEL
LIN {X 0,Y 378.956,Z 387.45,A -85,B 0,C 180,E1 -12275.312,E2 -12275.312} C_VEL
LIN {X 0,Y 378.756,Z 385.717,A -85,B 0,C 180,E1 -12278.8,E2 -12278.8} C_VEL
LIN {X 0,Y 378.761,Z 385.166,A -85,B 0,C 180,E1 -12281.912,E2 -12281.912} C_VEL
LIN {X 0,Y 378.945,Z 385.637,A -85,B 0,C 180,E1 -12284.81,E2 -12284.81} C_VEL
LIN {X 0,Y 379.38,Z 387.221,A -85,B 0,C 180,E1 -12287.817,E2 -12287.817} C_VEL
LIN {X 0,Y 380.079,Z 390.162,A -85,B 0,C 180,E1 -12290.952,E2 -12290.952} C_VEL
LIN {X 0,Y 381.172,Z 394.619,A -85,B 0,C 180,E1 -12294.22,E2 -12294.22} C_VEL
LIN {X 0,Y 382.088,Z 398.643,A -85,B 0,C 180,E1 -12296.508,E2 -12296.508} C_VEL
LIN {X 0,Y 382.956,Z 404.078,A -85,B 0,C 180,E1 -12299.079,E2 -12299.079} C_VEL
LIN {X 0,Y 382.694,Z 407.125,A -85,B 0,C 180,E1 -12300.274,E2 -12300.274} C_VEL
LIN {X 0,Y 380.004,Z 418.922,A -85,B 0,C 180,E1 -12304.238,E2 -12304.238} C_VEL
LIN {X 0,Y 378.283,Z 429.937,A -85,B 0,C 180,E1 -12307.613,E2 -12307.613} C_VEL
LIN {X 0,Y 377.111,Z 440.431,A -85,B 0,C 180,E1 -12310.629,E2 -12310.629} C_VEL
LIN {X 0,Y 379.312,Z 453.297,A -85,B 0,C 180,E1 -12311.283,E2 -12311.283} C_VEL
LIN {X 0,Y 380.11,Z 464.58,A -85,B 0,C 180,E1 -12311.955,E2 -12311.955} C_VEL
LIN {X 0,Y 380.026,Z 476.179,A -85,B 0,C 180,E1 -12312.788,E2 -12312.788} C_VEL
LIN {X 0,Y 378.87,Z 488.221,A -85,B 0,C 180,E1 -12313.844,E2 -12313.844} C_VEL
LIN {X 0,Y 377.879,Z 497.934,A -85,B 0,C 180,E1 -12314.907,E2 -12314.907} C_VEL
LIN {X 0,Y 376.918,Z 507.791,A -85,B 0,C 180,E1 -12316.247,E2 -12316.247} C_VEL
LIN {X 0,Y 376.119,Z 515.932,A -85,B 0,C 180,E1 -12317.591,E2 -12317.591} C_VEL
LIN {X 0,Y 375.396,Z 523.941,A -85,B 0,C 180,E1 -12319.209,E2 -12319.209} C_VEL
LIN {X 0,Y 375.018,Z 530.344,A -85,B 0,C 180,E1 -12320.834,E2 -12320.834} C_VEL
LIN {X 0,Y 374.86,Z 535.458,A -85,B 0,C 180,E1 -12322.459,E2 -12322.459} C_VEL
LIN {X 0,Y 374.783,Z 538.489,A -85,B 0,C 180,E1 -12323.652,E2 -12323.652} C_VEL
LIN {X 0,Y 374.783,Z 540.476,A -85,B 0,C 180,E1 -12324.62,E2 -12324.62} C_VEL
LIN {X 0,Y 374.766,Z 542.263,A -85,B 0,C 180,E1 -12325.698,E2 -12325.698} C_VEL
LIN {X 0,Y 374.921,Z 543.642,A -85,B 0,C 180,E1 -12326.776,E2 -12326.776} C_VEL
LIN {X 0,Y 374.985,Z 544.538,A -85,B 0,C 180,E1 -12327.852,E2 -12327.852} C_VEL
LIN {X 0,Y 374.923,Z 544.991,A -85,B 0,C 180,E1 -12328.926,E2 -12328.926} C_VEL
LIN {X 0,Y 374.891,Z 545.036,A -85,B 0,C 180,E1 -12330,E2 -12330} C_VEL
LIN {X 0,Y 374.922,Z 544.623,A -85,B 0,C 180,E1 -12331.074,E2 -12331.074} C_VEL
LIN {X 0,Y 375.032,Z 543.775,A -85,B 0,C 180,E1 -12332.148,E2 -12332.148} C_VEL
LIN {X 0,Y 374.981,Z 542.485,A -85,B 0,C 180,E1 -12333.223,E2 -12333.223} C_VEL
LIN {X 0,Y 374.829,Z 539.624,A -85,B 0,C 180,E1 -12334.84,E2 -12334.84} C_VEL
LIN {X 0,Y 374.923,Z 535.399,A -85,B 0,C 180,E1 -12336.537,E2 -12336.537} C_VEL
LIN {X 0,Y 375.011,Z 529.337,A -85,B 0,C 180,E1 -12338.351,E2 -12338.351} C_VEL
LIN {X 0,Y 375.199,Z 522.358,A -85,B 0,C 180,E1 -12339.978,E2 -12339.978} C_VEL
LIN {X 0,Y 375.707,Z 513.511,A -85,B 0,C 180,E1 -12341.601,E2 -12341.601} C_VEL
LIN {X 0,Y 376.288,Z 504.366,A -85,B 0,C 180,E1 -12342.951,E2 -12342.951} C_VEL
LIN {X 0,Y 376.771,Z 495.353,A -85,B 0,C 180,E1 -12344.033,E2 -12344.033} C_VEL
LIN {X 0,Y 377.471,Z 484.222,A -85,B 0,C 180,E1 -12345.109,E2 -12345.109} C_VEL
LIN {X 0,Y 378.102,Z 472.707,A -85,B 0,C 180,E1 -12345.981,E2 -12345.981} C_VEL
LIN {X 0,Y 377.866,Z 465.771,A -85,B 0,C 180,E1 -12346.408,E2 -12346.408} C_VEL
LIN {X 0,Y 376.816,Z 452.708,A -85,B 0,C 180,E1 -12347.048,E2 -12347.048} C_VEL
LIN {X 0,Y 376.04,Z 442.206,A -85,B 0,C 180,E1 -12347.399,E2 -12347.399} C_VEL
LIN {X 0,Y 376.975,Z 429.825,A -85,B 0,C 180,E1 -12350.745,E2 -12350.745} C_VEL
LIN {X 0,Y 378.225,Z 417.444,A -85,B 0,C 180,E1 -12354.129,E2 -12354.129} C_VEL
LIN {X 0,Y 379.875,Z 404.018,A -85,B 0,C 180,E1 -12357.849,E2 -12357.849} C_VEL
LIN {X 0,Y 380.699,Z 396.69,A -85,B 0,C 180,E1 -12359.897,E2 -12359.897} C_VEL
LIN {X 0,Y 378.976,Z 388.137,A -85,B 0,C 180,E1 -12362.534,E2 -12362.534} C_VEL
LIN {X 0,Y 376.77,Z 377.568,A -85,B 0,C 180,E1 -12365.933,E2 -12365.933} C_VEL
LIN {X 0,Y 376.001,Z 373.647,A -85,B 0,C 180,E1 -12367.238,E2 -12367.238} C_VEL
LIN {X 0,Y 375.942,Z 373.656,A -85,B 0,C 180,E1 -12370.867,E2 -12370.867} C_VEL
LIN {X 0,Y 375.956,Z 373.654,A -85,B 0,C 180,E1 -12374.736,E2 -12374.736} C_VEL
LIN {X 0,Y 375.945,Z 373.657,A -85,B 0,C 180,E1 -12378.397,E2 -12378.397} C_VEL
LIN {X 0,Y 375.977,Z 373.651,A -85,B 0,C 180,E1 -12381.729,E2 -12381.729} C_VEL
LIN {X 0,Y 375.981,Z 373.65,A -85,B 0,C 180,E1 -12385.332,E2 -12385.332} C_VEL
LIN {X 0,Y 375.958,Z 373.654,A -85,B 0,C 180,E1 -12388.438,E2 -12388.438} C_VEL
LIN {X 0,Y 375.984,Z 373.652,A -85,B 0,C 180,E1 -12392.14,E2 -12392.14} C_VEL
LIN {X 0,Y 376.007,Z 373.647,A -85,B 0,C 180,E1 -12394.539,E2 -12394.539} C_VEL
LIN {X 0,Y 375.964,Z 373.656,A -85,B 0,C 180,E1 -12398.046,E2 -12398.046} C_VEL
LIN {X 0,Y 376.025,Z 373.646,A -85,B 0,C 180,E1 -12401.474,E2 -12401.474} C_VEL
LIN {X 0,Y 376.06,Z 373.639,A -85,B 0,C 180,E1 -12404.833,E2 -12404.833} C_VEL
LIN {X 0,Y 376.051,Z 373.643,A -85,B 0,C 180,E1 -12408.137,E2 -12408.137} C_VEL
LIN {X 0,Y 376.258,Z 373.618,A -85,B 0,C 180,E1 -12411.877,E2 -12411.877} C_VEL
LIN {X 0,Y 376.173,Z 373.625,A -85,B 0,C 180,E1 -12414.64,E2 -12414.64} C_VEL
LIN {X 0,Y 376.355,Z 373.606,A -85,B 0,C 180,E1 -12417.86,E2 -12417.86} C_VEL
LIN {X 0,Y 376.49,Z 373.588,A -85,B 0,C 180,E1 -12420,E2 -12420} C_VEL
LIN {X 0,Y 376.186,Z 373.626,A -85,B 0,C 180,E1 -12423.213,E2 -12423.213} C_VEL
LIN {X 0,Y 376.235,Z 373.617,A -85,B 0,C 180,E1 -12426.634,E2 -12426.634} C_VEL
LIN {X 0,Y 376.207,Z 373.622,A -85,B 0,C 180,E1 -12428.595,E2 -12428.595} C_VEL
LIN {X 0,Y 376.06,Z 373.641,A -85,B 0,C 180,E1 -12431.863,E2 -12431.863} C_VEL
LIN {X 0,Y 376.061,Z 373.643,A -85,B 0,C 180,E1 -12435.167,E2 -12435.167} C_VEL
LIN {X 0,Y 376.01,Z 373.646,A -85,B 0,C 180,E1 -12438.527,E2 -12438.527} C_VEL
LIN {X 0,Y 375.964,Z 373.652,A -85,B 0,C 180,E1 -12441.954,E2 -12441.954} C_VEL
LIN {X 0,Y 376.007,Z 373.648,A -85,B 0,C 180,E1 -12445.461,E2 -12445.461} C_VEL
LIN {X 0,Y 375.971,Z 373.654,A -85,B 0,C 180,E1 -12449.079,E2 -12449.079} C_VEL
LIN {X 0,Y 375.952,Z 373.656,A -85,B 0,C 180,E1 -12452.828,E2 -12452.828} C_VEL
LIN {X 0,Y 375.959,Z 373.653,A -85,B 0,C 180,E1 -12455.416,E2 -12455.416} C_VEL
LIN {X 0,Y 375.976,Z 373.65,A -85,B 0,C 180,E1 -12458.271,E2 -12458.271} C_VEL
LIN {X 0,Y 375.935,Z 373.655,A -85,B 0,C 180,E1 -12461.601,E2 -12461.601} C_VEL
LIN {X 0,Y 375.93,Z 373.657,A -85,B 0,C 180,E1 -12465.268,E2 -12465.268} C_VEL
LIN {X 0,Y 375.937,Z 373.657,A -85,B 0,C 180,E1 -12468.399,E2 -12468.399} C_VEL
LIN {X 0,Y 375.976,Z 373.65,A -85,B 0,C 180,E1 -12471.73,E2 -12471.73} C_VEL
LIN {X 0,Y 375.981,Z 373.65,A -85,B 0,C 180,E1 -12475.333,E2 -12475.333} C_VEL
LIN {X 0,Y 375.959,Z 373.656,A -85,B 0,C 180,E1 -12478.438,E2 -12478.438} C_VEL
LIN {X 0,Y 375.985,Z 373.652,A -85,B 0,C 180,E1 -12482.141,E2 -12482.141} C_VEL
LIN {X 0,Y 376.008,Z 373.649,A -85,B 0,C 180,E1 -12484.539,E2 -12484.539} C_VEL
LIN {X 0,Y 375.973,Z 373.653,A -85,B 0,C 180,E1 -12488.047,E2 -12488.047} C_VEL
LIN {X 0,Y 376.032,Z 373.642,A -85,B 0,C 180,E1 -12491.475,E2 -12491.475} C_VEL
LIN {X 0,Y 376.064,Z 373.64,A -85,B 0,C 180,E1 -12494.833,E2 -12494.833} C_VEL
LIN {X 0,Y 376.053,Z 373.644,A -85,B 0,C 180,E1 -12498.137,E2 -12498.137} C_VEL
LIN {X 0,Y 376.221,Z 373.622,A -85,B 0,C 180,E1 -12501.919,E2 -12501.919} C_VEL
LIN {X 0,Y 376.172,Z 373.627,A -85,B 0,C 180,E1 -12504.64,E2 -12504.64} C_VEL
LIN {X 0,Y 376.355,Z 373.606,A -85,B 0,C 180,E1 -12507.86,E2 -12507.86} C_VEL
LIN {X 0,Y 376.492,Z 373.59,A -85,B 0,C 180,E1 -12510,E2 -12510} C_VEL
LIN {X 0,Y 376.188,Z 373.623,A -85,B 0,C 180,E1 -12513.213,E2 -12513.213} C_VEL
LIN {X 0,Y 376.242,Z 373.618,A -85,B 0,C 180,E1 -12516.435,E2 -12516.435} C_VEL
LIN {X 0,Y 376.122,Z 373.635,A -85,B 0,C 180,E1 -12519.682,E2 -12519.682} C_VEL
LIN {X 0,Y 376.092,Z 373.639,A -85,B 0,C 180,E1 -12523.658,E2 -12523.658} C_VEL
LIN {X 0,Y 376.047,Z 373.645,A -85,B 0,C 180,E1 -12527.608,E2 -12527.608} C_VEL
LIN {X 0,Y 375.981,Z 373.65,A -85,B 0,C 180,E1 -12530.832,E2 -12530.832} C_VEL
LIN {X 0,Y 375.996,Z 373.647,A -85,B 0,C 180,E1 -12534.282,E2 -12534.282} C_VEL
LIN {X 0,Y 376.022,Z 373.644,A -85,B 0,C 180,E1 -12536.652,E2 -12536.652} C_VEL
LIN {X 0,Y 375.967,Z 373.651,A -85,B 0,C 180,E1 -12540.313,E2 -12540.313} C_VEL
LIN {X 0,Y 375.962,Z 373.652,A -85,B 0,C 180,E1 -12544.112,E2 -12544.112} C_VEL
LIN {X 0,Y 375.956,Z 373.652,A -85,B 0,C 180,E1 -12546.741,E2 -12546.741} C_VEL
LIN {X 0,Y 375.986,Z 373.65,A -85,B 0,C 180,E1 -12550.028,E2 -12550.028} C_VEL
LIN {X 0,Y 375.253,Z 373.743,A -85,B 0,C 180,E1 -12550.922,E2 -12550.922} C_VEL
LIN {X 0,Y 372.346,Z 374.102,A -85,B 0,C 180,E1 -12552.374,E2 -12552.374} C_VEL
LIN {X 0,Y 369.943,Z 374.405,A -85,B 0,C 180,E1 -12553.548,E2 -12553.548} C_VEL
LIN {X 0,Y 368.948,Z 374.526,A -85,B 0,C 180,E1 -12554.457,E2 -12554.457} C_VEL
LIN {X 0,Y 368.884,Z 374.535,A -85,B 0,C 180,E1 -12554.764,E2 -12554.764} C_VEL
LIN {X 0,Y 368.885,Z 374.532,A -85,B 0,C 180,E1 -12558.178,E2 -12558.178} C_VEL
LIN {X 0,Y 368.913,Z 374.533,A -85,B 0,C 180,E1 -12561.359,E2 -12561.359} C_VEL
LIN {X 0,Y 368.94,Z 374.531,A -85,B 0,C 180,E1 -12565.147,E2 -12565.147} C_VEL
LIN {X 0,Y 369.137,Z 374.642,A -85,B 0,C 180,E1 -12568.81,E2 -12568.81} C_VEL
LIN {X 0,Y 369.128,Z 378.624,A -85,B 0,C 180,E1 -12571.142,E2 -12571.142} C_VEL
LIN {X 0,Y 368.747,Z 385.704,A -85,B 0,C 180,E1 -12575.209,E2 -12575.209} C_VEL
LIN {X 0,Y 368.455,Z 392.794,A -85,B 0,C 180,E1 -12579.171,E2 -12579.171} C_VEL
LIN {X 0,Y 368.248,Z 399.044,A -85,B 0,C 180,E1 -12582.603,E2 -12582.603} C_VEL
LIN {X 0,Y 368.056,Z 405.716,A -85,B 0,C 180,E1 -12586.191,E2 -12586.191} C_VEL
LIN {X 0,Y 367.97,Z 410.411,A -85,B 0,C 180,E1 -12588.675,E2 -12588.675} C_VEL
LIN {X 0,Y 369.234,Z 420.808,A -85,B 0,C 180,E1 -12589.305,E2 -12589.305} C_VEL
LIN {X 0,Y 369.901,Z 428.226,A -85,B 0,C 180,E1 -12589.878,E2 -12589.878} C_VEL
LIN {X 0,Y 369.437,Z 438.284,A -85,B 0,C 180,E1 -12590.832,E2 -12590.832} C_VEL
LIN {X 0,Y 369.055,Z 446.183,A -85,B 0,C 180,E1 -12591.789,E2 -12591.789} C_VEL
LIN {X 0,Y 368.867,Z 453.458,A -85,B 0,C 180,E1 -12592.886,E2 -12592.886} C_VEL
LIN {X 0,Y 368.582,Z 460.613,A -85,B 0,C 180,E1 -12594.255,E2 -12594.255} C_VEL
LIN {X 0,Y 368.375,Z 466.123,A -85,B 0,C 180,E1 -12595.623,E2 -12595.623} C_VEL
LIN {X 0,Y 368.042,Z 470.948,A -85,B 0,C 180,E1 -12597.264,E2 -12597.264} C_VEL
LIN {X 0,Y 367.928,Z 474.086,A -85,B 0,C 180,E1 -12598.905,E2 -12598.905} C_VEL
LIN {X 0,Y 367.908,Z 475.314,A -85,B 0,C 180,E1 -12600,E2 -12600} C_VEL
LIN {X 0,Y 367.972,Z 475.881,A -85,B 0,C 180,E1 -12601.094,E2 -12601.094} C_VEL
LIN {X 0,Y 368.122,Z 475.791,A -85,B 0,C 180,E1 -12602.188,E2 -12602.188} C_VEL
LIN {X 0,Y 368.385,Z 475.043,A -85,B 0,C 180,E1 -12603.281,E2 -12603.281} C_VEL
LIN {X 0,Y 369.11,Z 472.64,A -85,B 0,C 180,E1 -12604.915,E2 -12604.915} C_VEL
LIN {X 0,Y 369.715,Z 468.678,A -85,B 0,C 180,E1 -12606.549,E2 -12606.549} C_VEL
LIN {X 0,Y 370.579,Z 462.928,A -85,B 0,C 180,E1 -12608.177,E2 -12608.177} C_VEL
LIN {X 0,Y 371.504,Z 456.539,A -85,B 0,C 180,E1 -12609.528,E2 -12609.528} C_VEL
LIN {X 0,Y 372.542,Z 448.275,A -85,B 0,C 180,E1 -12610.874,E2 -12610.874} C_VEL
LIN {X 0,Y 373.647,Z 438.631,A -85,B 0,C 180,E1 -12612.079,E2 -12612.079} C_VEL
LIN {X 0,Y 373.851,Z 434.823,A -85,B 0,C 180,E1 -12612.485,E2 -12612.485} C_VEL
LIN {X 0,Y 372.194,Z 425.347,A -85,B 0,C 180,E1 -12613.521,E2 -12613.521} C_VEL
LIN {X 0,Y 369.325,Z 415.185,A -85,B 0,C 180,E1 -12614.512,E2 -12614.512} C_VEL
LIN {X 0,Y 369.806,Z 409.591,A -85,B 0,C 180,E1 -12618.152,E2 -12618.152} C_VEL
LIN {X 0,Y 370.324,Z 404.648,A -85,B 0,C 180,E1 -12621.577,E2 -12621.577} C_VEL
LIN {X 0,Y 370.943,Z 400.512,A -85,B 0,C 180,E1 -12624.634,E2 -12624.634} C_VEL
LIN {X 0,Y 371.756,Z 396.079,A -85,B 0,C 180,E1 -12628.205,E2 -12628.205} C_VEL
LIN {X 0,Y 372.217,Z 393.44,A -85,B 0,C 180,E1 -12630.651,E2 -12630.651} C_VEL
LIN {X 0,Y 372.318,Z 391.184,A -85,B 0,C 180,E1 -12633.19,E2 -12633.19} C_VEL
LIN {X 0,Y 372.171,Z 389.41,A -85,B 0,C 180,E1 -12635.831,E2 -12635.831} C_VEL
LIN {X 0,Y 372.067,Z 387.983,A -85,B 0,C 180,E1 -12639.244,E2 -12639.244} C_VEL
LIN {X 0,Y 372.074,Z 387.676,A -85,B 0,C 180,E1 -12641.384,E2 -12641.384} C_VEL
LIN {X 0,Y 372.26,Z 388.033,A -85,B 0,C 180,E1 -12644.31,E2 -12644.31} C_VEL
LIN {X 0,Y 372.665,Z 389.47,A -85,B 0,C 180,E1 -12647.349,E2 -12647.349} C_VEL
LIN {X 0,Y 373.245,Z 391.879,A -85,B 0,C 180,E1 -12650.193,E2 -12650.193} C_VEL
LIN {X 0,Y 374.055,Z 395.359,A -85,B 0,C 180,E1 -12653.041,E2 -12653.041} C_VEL
LIN {X 0,Y 375.16,Z 399.721,A -85,B 0,C 180,E1 -12655.805,E2 -12655.805} C_VEL
LIN {X 0,Y 376.046,Z 404.952,A -85,B 0,C 180,E1 -12658.446,E2 -12658.446} C_VEL
LIN {X 0,Y 376.11,Z 407.896,A -85,B 0,C 180,E1 -12659.7,E2 -12659.7} C_VEL
LIN {X 0,Y 374.093,Z 415.986,A -85,B 0,C 180,E1 -12662.595,E2 -12662.595} C_VEL
LIN {X 0,Y 372.055,Z 426.536,A -85,B 0,C 180,E1 -12666.038,E2 -12666.038} C_VEL
LIN {X 0,Y 370.507,Z 437.838,A -85,B 0,C 180,E1 -12669.456,E2 -12669.456} C_VEL
LIN {X 0,Y 370.26,Z 440.067,A -85,B 0,C 180,E1 -12670.101,E2 -12670.101} C_VEL
LIN {X 0,Y 372.632,Z 453.242,A -85,B 0,C 180,E1 -12670.821,E2 -12670.821} C_VEL
LIN {X 0,Y 373.494,Z 465.411,A -85,B 0,C 180,E1 -12671.591,E2 -12671.591} C_VEL
LIN {X 0,Y 373.287,Z 476.93,A -85,B 0,C 180,E1 -12672.468,E2 -12672.468} C_VEL
LIN {X 0,Y 372.085,Z 488.66,A -85,B 0,C 180,E1 -12673.541,E2 -12673.541} C_VEL
LIN {X 0,Y 370.911,Z 499.141,A -85,B 0,C 180,E1 -12674.758,E2 -12674.758} C_VEL
LIN {X 0,Y 369.807,Z 509.521,A -85,B 0,C 180,E1 -12676.257,E2 -12676.257} C_VEL
LIN {X 0,Y 368.919,Z 518.587,A -85,B 0,C 180,E1 -12677.904,E2 -12677.904} C_VEL
LIN {X 0,Y 368.189,Z 525.918,A -85,B 0,C 180,E1 -12679.552,E2 -12679.552} C_VEL
LIN {X 0,Y 367.88,Z 531.785,A -85,B 0,C 180,E1 -12681.209,E2 -12681.209} C_VEL
LIN {X 0,Y 367.752,Z 536.411,A -85,B 0,C 180,E1 -12682.864,E2 -12682.864} C_VEL
LIN {X 0,Y 367.701,Z 539.915,A -85,B 0,C 180,E1 -12684.516,E2 -12684.516} C_VEL
LIN {X 0,Y 367.686,Z 541.674,A -85,B 0,C 180,E1 -12685.615,E2 -12685.615} C_VEL
LIN {X 0,Y 367.834,Z 543.009,A -85,B 0,C 180,E1 -12686.714,E2 -12686.714} C_VEL
LIN {X 0,Y 367.908,Z 543.861,A -85,B 0,C 180,E1 -12687.81,E2 -12687.81} C_VEL
LIN {X 0,Y 367.876,Z 544.29,A -85,B 0,C 180,E1 -12688.905,E2 -12688.905} C_VEL
LIN {X 0,Y 367.842,Z 544.296,A -85,B 0,C 180,E1 -12690,E2 -12690} C_VEL
LIN {X 0,Y 367.876,Z 543.83,A -85,B 0,C 180,E1 -12691.094,E2 -12691.094} C_VEL
LIN {X 0,Y 367.984,Z 542.95,A -85,B 0,C 180,E1 -12692.189,E2 -12692.189} C_VEL
LIN {X 0,Y 367.914,Z 541.608,A -85,B 0,C 180,E1 -12693.285,E2 -12693.285} C_VEL
LIN {X 0,Y 367.773,Z 538.657,A -85,B 0,C 180,E1 -12694.933,E2 -12694.933} C_VEL
LIN {X 0,Y 367.845,Z 534.565,A -85,B 0,C 180,E1 -12696.582,E2 -12696.582} C_VEL
LIN {X 0,Y 367.941,Z 528.168,A -85,B 0,C 180,E1 -12698.513,E2 -12698.513} C_VEL
LIN {X 0,Y 368.163,Z 521.013,A -85,B 0,C 180,E1 -12700.17,E2 -12700.17} C_VEL
LIN {X 0,Y 368.685,Z 512.023,A -85,B 0,C 180,E1 -12701.825,E2 -12701.825} C_VEL
LIN {X 0,Y 369.33,Z 502.625,A -85,B 0,C 180,E1 -12703.2,E2 -12703.2} C_VEL
LIN {X 0,Y 369.722,Z 494.926,A -85,B 0,C 180,E1 -12704.135,E2 -12704.135} C_VEL
LIN {X 0,Y 370.449,Z 483.49,A -85,B 0,C 180,E1 -12705.262,E2 -12705.262} C_VEL
LIN {X 0,Y 371.094,Z 471.922,A -85,B 0,C 180,E1 -12706.15,E2 -12706.15} C_VEL
LIN {X 0,Y 370.294,Z 459.252,A -85,B 0,C 180,E1 -12706.895,E2 -12706.895} C_VEL
LIN {X 0,Y 369.29,Z 446.698,A -85,B 0,C 180,E1 -12707.424,E2 -12707.424} C_VEL
LIN {X 0,Y 369.001,Z 441.901,A -85,B 0,C 180,E1 -12707.599,E2 -12707.599} C_VEL
LIN {X 0,Y 370.017,Z 429.036,A -85,B 0,C 180,E1 -12711.154,E2 -12711.154} C_VEL
LIN {X 0,Y 371.421,Z 416.255,A -85,B 0,C 180,E1 -12714.735,E2 -12714.735} C_VEL
LIN {X 0,Y 373.238,Z 402.283,A -85,B 0,C 180,E1 -12718.696,E2 -12718.696} C_VEL
LIN {X 0,Y 373.673,Z 397.471,A -85,B 0,C 180,E1 -12720.098,E2 -12720.098} C_VEL
LIN {X 0,Y 371.629,Z 387.462,A -85,B 0,C 180,E1 -12723.259,E2 -12723.259} C_VEL
LIN {X 0,Y 369.316,Z 376.375,A -85,B 0,C 180,E1 -12726.941,E2 -12726.941} C_VEL
LIN {X 0,Y 368.944,Z 374.527,A -85,B 0,C 180,E1 -12727.644,E2 -12727.644} C_VEL
LIN {X 0,Y 368.912,Z 374.534,A -85,B 0,C 180,E1 -12730.37,E2 -12730.37} C_VEL
LIN {X 0,Y 368.885,Z 374.534,A -85,B 0,C 180,E1 -12733.616,E2 -12733.616} C_VEL
LIN {X 0,Y 368.887,Z 374.535,A -85,B 0,C 180,E1 -12736.696,E2 -12736.696} C_VEL
LIN {X 0,Y 368.936,Z 374.527,A -85,B 0,C 180,E1 -12739.638,E2 -12739.638} C_VEL
LIN {X 0,Y 368.904,Z 374.531,A -85,B 0,C 180,E1 -12743.144,E2 -12743.144} C_VEL
LIN {X 0,Y 368.899,Z 374.534,A -85,B 0,C 180,E1 -12746.462,E2 -12746.462} C_VEL
LIN {X 0,Y 368.929,Z 374.527,A -85,B 0,C 180,E1 -12749.046,E2 -12749.046} C_VEL
LIN {X 0,Y 368.964,Z 374.523,A -85,B 0,C 180,E1 -12752.797,E2 -12752.797} C_VEL
LIN {X 0,Y 368.946,Z 374.529,A -85,B 0,C 180,E1 -12756.113,E2 -12756.113} C_VEL
LIN {X 0,Y 368.938,Z 374.531,A -85,B 0,C 180,E1 -12759.947,E2 -12759.947} C_VEL
LIN {X 0,Y 368.977,Z 374.523,A -85,B 0,C 180,E1 -12763.399,E2 -12763.399} C_VEL
LIN {X 0,Y 369.058,Z 374.512,A -85,B 0,C 180,E1 -12766.79,E2 -12766.79} C_VEL
LIN {X 0,Y 369.068,Z 374.512,A -85,B 0,C 180,E1 -12770.132,E2 -12770.132} C_VEL
LIN {X 0,Y 369.189,Z 374.495,A -85,B 0,C 180,E1 -12772.342,E2 -12772.342} C_VEL
LIN {X 0,Y 369.146,Z 374.5,A -85,B 0,C 180,E1 -12774.538,E2 -12774.538} C_VEL
LIN {X 0,Y 369.32,Z 374.482,A -85,B 0,C 180,E1 -12777.819,E2 -12777.819} C_VEL
LIN {X 0,Y 369.46,Z 374.463,A -85,B 0,C 180,E1 -12780,E2 -12780} C_VEL
LIN {X 0,Y 369.318,Z 374.479,A -85,B 0,C 180,E1 -12782.181,E2 -12782.181} C_VEL
LIN {X 0,Y 369.205,Z 374.493,A -85,B 0,C 180,E1 -12786.622,E2 -12786.622} C_VEL
LIN {X 0,Y 369.14,Z 374.502,A -85,B 0,C 180,E1 -12788.761,E2 -12788.761} C_VEL
LIN {X 0,Y 369.014,Z 374.517,A -85,B 0,C 180,E1 -12792.093,E2 -12792.093} C_VEL
LIN {X 0,Y 369,Z 374.522,A -85,B 0,C 180,E1 -12795.465,E2 -12795.465} C_VEL
LIN {X 0,Y 368.959,Z 374.527,A -85,B 0,C 180,E1 -12798.894,E2 -12798.894} C_VEL
LIN {X 0,Y 368.933,Z 374.528,A -85,B 0,C 180,E1 -12802.395,E2 -12802.395} C_VEL
LIN {X 0,Y 369.001,Z 374.518,A -85,B 0,C 180,E1 -12805.98,E2 -12805.98} C_VEL
LIN {X 0,Y 368.96,Z 374.527,A -85,B 0,C 180,E1 -12808.811,E2 -12808.811} C_VEL
LIN {X 0,Y 368.899,Z 374.532,A -85,B 0,C 180,E1 -12812.238,E2 -12812.238} C_VEL
LIN {X 0,Y 368.93,Z 374.532,A -85,B 0,C 180,E1 -12815.002,E2 -12815.002} C_VEL
LIN {X 0,Y 368.911,Z 374.533,A -85,B 0,C 180,E1 -12818.641,E2 -12818.641} C_VEL
LIN {X 0,Y 368.882,Z 374.534,A -85,B 0,C 180,E1 -12822.01,E2 -12822.01} C_VEL
LIN {X 0,Y 368.887,Z 374.535,A -85,B 0,C 180,E1 -12825.177,E2 -12825.177} C_VEL
LIN {X 0,Y 368.885,Z 374.534,A -85,B 0,C 180,E1 -12828.178,E2 -12828.178} C_VEL
LIN {X 0,Y 368.91,Z 374.53,A -85,B 0,C 180,E1 -12831.36,E2 -12831.36} C_VEL
LIN {X 0,Y 368.938,Z 374.528,A -85,B 0,C 180,E1 -12835.147,E2 -12835.147} C_VEL
LIN {X 0,Y 368.93,Z 374.528,A -85,B 0,C 180,E1 -12839.047,E2 -12839.047} C_VEL
LIN {X 0,Y 368.965,Z 374.526,A -85,B 0,C 180,E1 -12842.797,E2 -12842.797} C_VEL
LIN {X 0,Y 368.947,Z 374.529,A -85,B 0,C 180,E1 -12846.113,E2 -12846.113} C_VEL
LIN {X 0,Y 368.947,Z 374.527,A -85,B 0,C 180,E1 -12849.948,E2 -12849.948} C_VEL
LIN {X 0,Y 368.981,Z 374.521,A -85,B 0,C 180,E1 -12853.399,E2 -12853.399} C_VEL
LIN {X 0,Y 369.06,Z 374.513,A -85,B 0,C 180,E1 -12856.79,E2 -12856.79} C_VEL
LIN {X 0,Y 369.072,Z 374.514,A -85,B 0,C 180,E1 -12860.132,E2 -12860.132} C_VEL
LIN {X 0,Y 369.164,Z 374.501,A -85,B 0,C 180,E1 -12862.342,E2 -12862.342} C_VEL
LIN {X 0,Y 369.145,Z 374.503,A -85,B 0,C 180,E1 -12864.538,E2 -12864.538} C_VEL
LIN {X 0,Y 369.32,Z 374.483,A -85,B 0,C 180,E1 -12867.819,E2 -12867.819} C_VEL
LIN {X 0,Y 369.462,Z 374.465,A -85,B 0,C 180,E1 -12870,E2 -12870} C_VEL
LIN {X 0,Y 369.319,Z 374.482,A -85,B 0,C 180,E1 -12872.181,E2 -12872.181} C_VEL
LIN {X 0,Y 369.202,Z 374.494,A -85,B 0,C 180,E1 -12876.559,E2 -12876.559} C_VEL
LIN {X 0,Y 369.071,Z 374.514,A -85,B 0,C 180,E1 -12879.868,E2 -12879.868} C_VEL
LIN {X 0,Y 369.04,Z 374.519,A -85,B 0,C 180,E1 -12883.773,E2 -12883.773} C_VEL
LIN {X 0,Y 369.004,Z 374.522,A -85,B 0,C 180,E1 -12887.768,E2 -12887.768} C_VEL
LIN {X 0,Y 368.932,Z 374.53,A -85,B 0,C 180,E1 -12891.22,E2 -12891.22} C_VEL
LIN {X 0,Y 368.96,Z 374.523,A -85,B 0,C 180,E1 -12894.775,E2 -12894.775} C_VEL
LIN {X 0,Y 368.966,Z 374.526,A -85,B 0,C 180,E1 -12897.204,E2 -12897.204} C_VEL
LIN {X 0,Y 368.932,Z 374.529,A -85,B 0,C 180,E1 -12900.954,E2 -12900.954} C_VEL
LIN {X 0,Y 368.932,Z 374.529,A -85,B 0,C 180,E1 -12905.002,E2 -12905.002} C_VEL
LIN {X 0,Y 368.911,Z 374.53,A -85,B 0,C 180,E1 -12908.64,E2 -12908.64} C_VEL
LIN {X 0,Y 368.884,Z 374.534,A -85,B 0,C 180,E1 -12912.01,E2 -12912.01} C_VEL
LIN {X 0,Y 368.884,Z 374.535,A -85,B 0,C 180,E1 -12914.764,E2 -12914.764} C_VEL
LIN {X 0,Y 368.258,Z 374.618,A -85,B 0,C 180,E1 -12915.676,E2 -12915.676} C_VEL
LIN {X 0,Y 365.4,Z 374.978,A -85,B 0,C 180,E1 -12917.157,E2 -12917.157} C_VEL
LIN {X 0,Y 362.957,Z 375.279,A -85,B 0,C 180,E1 -12918.355,E2 -12918.355} C_VEL
LIN {X 0,Y 361.915,Z 375.405,A -85,B 0,C 180,E1 -12919.282,E2 -12919.282} C_VEL
LIN {X 0,Y 361.836,Z 375.412,A -85,B 0,C 180,E1 -12919.596,E2 -12919.596} C_VEL
LIN {X 0,Y 361.872,Z 375.411,A -85,B 0,C 180,E1 -12922.982,E2 -12922.982} C_VEL
LIN {X 0,Y 361.889,Z 375.406,A -85,B 0,C 180,E1 -12926.624,E2 -12926.624} C_VEL
LIN {X 0,Y 362.043,Z 375.394,A -85,B 0,C 180,E1 -12928.664,E2 -12928.664} C_VEL
LIN {X 0,Y 362.102,Z 379.244,A -85,B 0,C 180,E1 -12930.973,E2 -12930.973} C_VEL
LIN {X 0,Y 361.707,Z 385.666,A -85,B 0,C 180,E1 -12934.693,E2 -12934.693} C_VEL
LIN {X 0,Y 361.439,Z 392.062,A -85,B 0,C 180,E1 -12938.318,E2 -12938.318} C_VEL
LIN {X 0,Y 361.249,Z 397.341,A -85,B 0,C 180,E1 -12941.276,E2 -12941.276} C_VEL
LIN {X 0,Y 361.06,Z 403.693,A -85,B 0,C 180,E1 -12944.765,E2 -12944.765} C_VEL
LIN {X 0,Y 360.913,Z 410.664,A -85,B 0,C 180,E1 -12948.522,E2 -12948.522} C_VEL
LIN {X 0,Y 362.244,Z 421.93,A -85,B 0,C 180,E1 -12949.238,E2 -12949.238} C_VEL
LIN {X 0,Y 362.82,Z 429.213,A -85,B 0,C 180,E1 -12949.819,E2 -12949.819} C_VEL
LIN {X 0,Y 362.36,Z 439.165,A -85,B 0,C 180,E1 -12950.793,E2 -12950.793} C_VEL
LIN {X 0,Y 361.95,Z 448.017,A -85,B 0,C 180,E1 -12951.908,E2 -12951.908} C_VEL
LIN {X 0,Y 361.782,Z 455.169,A -85,B 0,C 180,E1 -12953.048,E2 -12953.048} C_VEL
LIN {X 0,Y 361.459,Z 462.009,A -85,B 0,C 180,E1 -12954.421,E2 -12954.421} C_VEL
LIN {X 0,Y 361.302,Z 466.406,A -85,B 0,C 180,E1 -12955.537,E2 -12955.537} C_VEL
LIN {X 0,Y 360.972,Z 471.357,A -85,B 0,C 180,E1 -12957.21,E2 -12957.21} C_VEL
LIN {X 0,Y 360.878,Z 474.626,A -85,B 0,C 180,E1 -12958.884,E2 -12958.884} C_VEL
LIN {X 0,Y 360.856,Z 475.954,A -85,B 0,C 180,E1 -12960,E2 -12960} C_VEL
LIN {X 0,Y 360.922,Z 476.619,A -85,B 0,C 180,E1 -12961.116,E2 -12961.116} C_VEL
LIN {X 0,Y 361.079,Z 476.619,A -85,B 0,C 180,E1 -12962.231,E2 -12962.231} C_VEL
LIN {X 0,Y 361.356,Z 475.956,A -85,B 0,C 180,E1 -12963.345,E2 -12963.345} C_VEL
LIN {X 0,Y 361.782,Z 474.622,A -85,B 0,C 180,E1 -12964.457,E2 -12964.457} C_VEL
LIN {X 0,Y 362.541,Z 471.374,A -85,B 0,C 180,E1 -12966.12,E2 -12966.12} C_VEL
LIN {X 0,Y 363.371,Z 466.487,A -85,B 0,C 180,E1 -12967.781,E2 -12967.781} C_VEL
LIN {X 0,Y 364.262,Z 460.92,A -85,B 0,C 180,E1 -12969.159,E2 -12969.159} C_VEL
LIN {X 0,Y 365.266,Z 454.062,A -85,B 0,C 180,E1 -12970.473,E2 -12970.473} C_VEL
LIN {X 0,Y 366.478,Z 445.259,A -85,B 0,C 180,E1 -12971.79,E2 -12971.79} C_VEL
LIN {X 0,Y 367.347,Z 436.694,A -85,B 0,C 180,E1 -12972.808,E2 -12972.808} C_VEL
LIN {X 0,Y 365.771,Z 427.275,A -85,B 0,C 180,E1 -12973.898,E2 -12973.898} C_VEL
LIN {X 0,Y 362.427,Z 415.7,A -85,B 0,C 180,E1 -12975.137,E2 -12975.137} C_VEL
LIN {X 0,Y 363.045,Z 409.662,A -85,B 0,C 180,E1 -12979.214,E2 -12979.214} C_VEL
LIN {X 0,Y 363.609,Z 404.79,A -85,B 0,C 180,E1 -12982.741,E2 -12982.741} C_VEL
LIN {X 0,Y 364.444,Z 400.266,A -85,B 0,C 180,E1 -12986.33,E2 -12986.33} C_VEL
LIN {X 0,Y 365.048,Z 397.468,A -85,B 0,C 180,E1 -12988.771,E2 -12988.771} C_VEL
LIN {X 0,Y 365.459,Z 394.934,A -85,B 0,C 180,E1 -12991.281,E2 -12991.281} C_VEL
LIN {X 0,Y 365.534,Z 392.646,A -85,B 0,C 180,E1 -12994.234,E2 -12994.234} C_VEL
LIN {X 0,Y 365.426,Z 391.318,A -85,B 0,C 180,E1 -12996.599,E2 -12996.599} C_VEL
LIN {X 0,Y 365.404,Z 390.306,A -85,B 0,C 180,E1 -12999.705,E2 -12999.705} C_VEL
LIN {X 0,Y 365.541,Z 390.28,A -85,B 0,C 180,E1 -13003.063,E2 -13003.063} C_VEL
LIN {X 0,Y 365.839,Z 391.383,A -85,B 0,C 180,E1 -13006.244,E2 -13006.244} C_VEL
LIN {X 0,Y 366.429,Z 393.586,A -85,B 0,C 180,E1 -13009.299,E2 -13009.299} C_VEL
LIN {X 0,Y 367.171,Z 396.801,A -85,B 0,C 180,E1 -13012.228,E2 -13012.228} C_VEL
LIN {X 0,Y 368.241,Z 401.047,A -85,B 0,C 180,E1 -13015.152,E2 -13015.152} C_VEL
LIN {X 0,Y 369.109,Z 405.872,A -85,B 0,C 180,E1 -13017.782,E2 -13017.782} C_VEL
LIN {X 0,Y 369.446,Z 408.684,A -85,B 0,C 180,E1 -13019.094,E2 -13019.094} C_VEL
LIN {X 0,Y 368.834,Z 411.739,A -85,B 0,C 180,E1 -13020.302,E2 -13020.302} C_VEL
LIN {X 0,Y 366.367,Z 421.614,A -85,B 0,C 180,E1 -13023.819,E2 -13023.819} C_VEL
LIN {X 0,Y 364.196,Z 434.163,A -85,B 0,C 180,E1 -13027.861,E2 -13027.861} C_VEL
LIN {X 0,Y 363.485,Z 439.822,A -85,B 0,C 180,E1 -13029.54,E2 -13029.54} C_VEL
LIN {X 0,Y 365.814,Z 452.055,A -85,B 0,C 180,E1 -13030.254,E2 -13030.254} C_VEL
LIN {X 0,Y 366.844,Z 464.075,A -85,B 0,C 180,E1 -13031.049,E2 -13031.049} C_VEL
LIN {X 0,Y 366.731,Z 476.272,A -85,B 0,C 180,E1 -13032.007,E2 -13032.007} C_VEL
LIN {X 0,Y 365.444,Z 487.879,A -85,B 0,C 180,E1 -13033.089,E2 -13033.089} C_VEL
LIN {X 0,Y 364.194,Z 498.331,A -85,B 0,C 180,E1 -13034.326,E2 -13034.326} C_VEL
LIN {X 0,Y 363.079,Z 507.841,A -85,B 0,C 180,E1 -13035.713,E2 -13035.713} C_VEL
LIN {X 0,Y 362.193,Z 515.695,A -85,B 0,C 180,E1 -13037.106,E2 -13037.106} C_VEL
LIN {X 0,Y 361.375,Z 523.38,A -85,B 0,C 180,E1 -13038.785,E2 -13038.785} C_VEL
LIN {X 0,Y 360.913,Z 529.608,A -85,B 0,C 180,E1 -13040.472,E2 -13040.472} C_VEL
LIN {X 0,Y 360.689,Z 534.555,A -85,B 0,C 180,E1 -13042.16,E2 -13042.16} C_VEL
LIN {X 0,Y 360.626,Z 538.003,A -85,B 0,C 180,E1 -13043.673,E2 -13043.673} C_VEL
LIN {X 0,Y 360.608,Z 541.096,A -85,B 0,C 180,E1 -13045.529,E2 -13045.529} C_VEL
LIN {X 0,Y 360.751,Z 542.362,A -85,B 0,C 180,E1 -13046.649,E2 -13046.649} C_VEL
LIN {X 0,Y 360.832,Z 543.185,A -85,B 0,C 180,E1 -13047.767,E2 -13047.767} C_VEL
LIN {X 0,Y 360.829,Z 543.587,A -85,B 0,C 180,E1 -13048.884,E2 -13048.884} C_VEL
LIN {X 0,Y 360.794,Z 543.525,A -85,B 0,C 180,E1 -13050,E2 -13050} C_VEL
LIN {X 0,Y 360.83,Z 543.022,A -85,B 0,C 180,E1 -13051.116,E2 -13051.116} C_VEL
LIN {X 0,Y 360.937,Z 542.109,A -85,B 0,C 180,E1 -13052.232,E2 -13052.232} C_VEL
LIN {X 0,Y 360.85,Z 540.689,A -85,B 0,C 180,E1 -13053.349,E2 -13053.349} C_VEL
LIN {X 0,Y 360.72,Z 537.655,A -85,B 0,C 180,E1 -13055.03,E2 -13055.03} C_VEL
LIN {X 0,Y 360.779,Z 533.47,A -85,B 0,C 180,E1 -13056.712,E2 -13056.712} C_VEL
LIN {X 0,Y 360.862,Z 527.983,A -85,B 0,C 180,E1 -13058.399,E2 -13058.399} C_VEL
LIN {X 0,Y 361.073,Z 520.99,A -85,B 0,C 180,E1 -13060.089,E2 -13060.089} C_VEL
LIN {X 0,Y 361.587,Z 512.126,A -85,B 0,C 180,E1 -13061.776,E2 -13061.776} C_VEL
LIN {X 0,Y 362.197,Z 502.937,A -85,B 0,C 180,E1 -13063.179,E2 -13063.179} C_VEL
LIN {X 0,Y 362.636,Z 494.771,A -85,B 0,C 180,E1 -13064.203,E2 -13064.203} C_VEL
LIN {X 0,Y 363.352,Z 484.235,A -85,B 0,C 180,E1 -13065.28,E2 -13065.28} C_VEL
LIN {X 0,Y 364.049,Z 472.069,A -85,B 0,C 180,E1 -13066.255,E2 -13066.255} C_VEL
LIN {X 0,Y 363.257,Z 459.889,A -85,B 0,C 180,E1 -13067.002,E2 -13067.002} C_VEL
LIN {X 0,Y 362.246,Z 446.711,A -85,B 0,C 180,E1 -13067.581,E2 -13067.581} C_VEL
LIN {X 0,Y 361.957,Z 441.634,A -85,B 0,C 180,E1 -13067.761,E2 -13067.761} C_VEL
LIN {X 0,Y 363.33,Z 426.2,A -85,B 0,C 180,E1 -13072.163,E2 -13072.163} C_VEL
LIN {X 0,Y 365.037,Z 411.896,A -85,B 0,C 180,E1 -13076.284,E2 -13076.284} C_VEL
LIN {X 0,Y 366.572,Z 400.554,A -85,B 0,C 180,E1 -13079.583,E2 -13079.583} C_VEL
LIN {X 0,Y 366.351,Z 396.82,A -85,B 0,C 180,E1 -13080.734,E2 -13080.734} C_VEL
LIN {X 0,Y 364.027,Z 385.683,A -85,B 0,C 180,E1 -13084.382,E2 -13084.382} C_VEL
LIN {X 0,Y 361.897,Z 375.404,A -85,B 0,C 180,E1 -13087.959,E2 -13087.959} C_VEL
LIN {X 0,Y 361.828,Z 375.415,A -85,B 0,C 180,E1 -13091.33,E2 -13091.33} C_VEL
LIN {X 0,Y 361.848,Z 375.414,A -85,B 0,C 180,E1 -13094.363,E2 -13094.363} C_VEL
LIN {X 0,Y 361.841,Z 375.411,A -85,B 0,C 180,E1 -13097.567,E2 -13097.567} C_VEL
LIN {X 0,Y 361.873,Z 375.406,A -85,B 0,C 180,E1 -13100.973,E2 -13100.973} C_VEL
LIN {X 0,Y 361.875,Z 375.407,A -85,B 0,C 180,E1 -13104.655,E2 -13104.655} C_VEL
LIN {X 0,Y 361.838,Z 375.413,A -85,B 0,C 180,E1 -13108.371,E2 -13108.371} C_VEL
LIN {X 0,Y 361.909,Z 375.405,A -85,B 0,C 180,E1 -13112.221,E2 -13112.221} C_VEL
LIN {X 0,Y 361.929,Z 375.4,A -85,B 0,C 180,E1 -13114.71,E2 -13114.71} C_VEL
LIN {X 0,Y 361.893,Z 375.406,A -85,B 0,C 180,E1 -13118.347,E2 -13118.347} C_VEL
LIN {X 0,Y 361.968,Z 375.397,A -85,B 0,C 180,E1 -13122.061,E2 -13122.061} C_VEL
LIN {X 0,Y 361.998,Z 375.393,A -85,B 0,C 180,E1 -13126.101,E2 -13126.101} C_VEL
LIN {X 0,Y 362.032,Z 375.39,A -85,B 0,C 180,E1 -13129.938,E2 -13129.938} C_VEL
LIN {X 0,Y 362.152,Z 375.372,A -85,B 0,C 180,E1 -13132.193,E2 -13132.193} C_VEL
LIN {X 0,Y 362.119,Z 375.375,A -85,B 0,C 180,E1 -13134.431,E2 -13134.431} C_VEL
LIN {X 0,Y 362.284,Z 375.359,A -85,B 0,C 180,E1 -13137.776,E2 -13137.776} C_VEL
LIN {X 0,Y 362.429,Z 375.339,A -85,B 0,C 180,E1 -13140,E2 -13140} C_VEL
LIN {X 0,Y 362.282,Z 375.355,A -85,B 0,C 180,E1 -13142.224,E2 -13142.224} C_VEL
LIN {X 0,Y 362.173,Z 375.369,A -85,B 0,C 180,E1 -13146.686,E2 -13146.686} C_VEL
LIN {X 0,Y 362.077,Z 375.383,A -85,B 0,C 180,E1 -13148.933,E2 -13148.933} C_VEL
LIN {X 0,Y 361.968,Z 375.394,A -85,B 0,C 180,E1 -13152.332,E2 -13152.332} C_VEL
LIN {X 0,Y 361.963,Z 375.395,A -85,B 0,C 180,E1 -13154.62,E2 -13154.62} C_VEL
LIN {X 0,Y 361.956,Z 375.396,A -85,B 0,C 180,E1 -13158.1,E2 -13158.1} C_VEL
LIN {X 0,Y 361.893,Z 375.406,A -85,B 0,C 180,E1 -13161.653,E2 -13161.653} C_VEL
LIN {X 0,Y 361.929,Z 375.403,A -85,B 0,C 180,E1 -13165.29,E2 -13165.29} C_VEL
LIN {X 0,Y 361.915,Z 375.401,A -85,B 0,C 180,E1 -13167.779,E2 -13167.779} C_VEL
LIN {X 0,Y 361.847,Z 375.413,A -85,B 0,C 180,E1 -13171.285,E2 -13171.285} C_VEL
LIN {X 0,Y 361.856,Z 375.409,A -85,B 0,C 180,E1 -13174.28,E2 -13174.28} C_VEL
LIN {X 0,Y 361.866,Z 375.409,A -85,B 0,C 180,E1 -13177.223,E2 -13177.223} C_VEL
LIN {X 0,Y 361.837,Z 375.415,A -85,B 0,C 180,E1 -13180.756,E2 -13180.756} C_VEL
LIN {X 0,Y 361.847,Z 375.412,A -85,B 0,C 180,E1 -13184.364,E2 -13184.364} C_VEL
LIN {X 0,Y 361.838,Z 375.41,A -85,B 0,C 180,E1 -13187.568,E2 -13187.568} C_VEL
LIN {X 0,Y 361.871,Z 375.409,A -85,B 0,C 180,E1 -13190.973,E2 -13190.973} C_VEL
LIN {X 0,Y 361.875,Z 375.41,A -85,B 0,C 180,E1 -13194.655,E2 -13194.655} C_VEL
LIN {X 0,Y 361.839,Z 375.414,A -85,B 0,C 180,E1 -13198.371,E2 -13198.371} C_VEL
LIN {X 0,Y 361.91,Z 375.405,A -85,B 0,C 180,E1 -13202.221,E2 -13202.221} C_VEL
LIN {X 0,Y 361.93,Z 375.403,A -85,B 0,C 180,E1 -13204.71,E2 -13204.71} C_VEL
LIN {X 0,Y 361.901,Z 375.407,A -85,B 0,C 180,E1 -13208.348,E2 -13208.348} C_VEL
LIN {X 0,Y 361.97,Z 375.397,A -85,B 0,C 180,E1 -13212.061,E2 -13212.061} C_VEL
LIN {X 0,Y 362,Z 375.395,A -85,B 0,C 180,E1 -13216.101,E2 -13216.101} C_VEL
LIN {X 0,Y 362.036,Z 375.389,A -85,B 0,C 180,E1 -13219.938,E2 -13219.938} C_VEL
LIN {X 0,Y 362.163,Z 375.37,A -85,B 0,C 180,E1 -13223.314,E2 -13223.314} C_VEL
LIN {X 0,Y 362.284,Z 375.359,A -85,B 0,C 180,E1 -13227.777,E2 -13227.777} C_VEL
LIN {X 0,Y 362.431,Z 375.341,A -85,B 0,C 180,E1 -13230,E2 -13230} C_VEL
LIN {X 0,Y 362.283,Z 375.358,A -85,B 0,C 180,E1 -13232.224,E2 -13232.224} C_VEL
LIN {X 0,Y 362.164,Z 375.37,A -85,B 0,C 180,E1 -13236.687,E2 -13236.687} C_VEL
LIN {X 0,Y 362.035,Z 375.39,A -85,B 0,C 180,E1 -13240.062,E2 -13240.062} C_VEL
LIN {X 0,Y 362.001,Z 375.394,A -85,B 0,C 180,E1 -13243.899,E2 -13243.899} C_VEL
LIN {X 0,Y 361.97,Z 375.398,A -85,B 0,C 180,E1 -13247.939,E2 -13247.939} C_VEL
LIN {X 0,Y 361.895,Z 375.408,A -85,B 0,C 180,E1 -13251.653,E2 -13251.653} C_VEL
LIN {X 0,Y 361.931,Z 375.402,A -85,B 0,C 180,E1 -13255.29,E2 -13255.29} C_VEL
LIN {X 0,Y 361.911,Z 375.405,A -85,B 0,C 180,E1 -13257.779,E2 -13257.779} C_VEL
LIN {X 0,Y 361.84,Z 375.415,A -85,B 0,C 180,E1 -13261.629,E2 -13261.629} C_VEL
LIN {X 0,Y 361.877,Z 375.41,A -85,B 0,C 180,E1 -13265.345,E2 -13265.345} C_VEL
LIN {X 0,Y 361.873,Z 375.409,A -85,B 0,C 180,E1 -13269.027,E2 -13269.027} C_VEL
LIN {X 0,Y 361.839,Z 375.413,A -85,B 0,C 180,E1 -13272.829,E2 -13272.829} C_VEL
LIN {X 0,Y 361.838,Z 375.411,A -85,B 0,C 180,E1 -13275.944,E2 -13275.944} C_VEL
LIN {X 0,Y 361.836,Z 375.412,A -85,B 0,C 180,E1 -13279.596,E2 -13279.596} C_VEL
LIN {X 0,Y 361.188,Z 375.494,A -85,B 0,C 180,E1 -13280.525,E2 -13280.525} C_VEL
LIN {X 0,Y 358.357,Z 375.844,A -85,B 0,C 180,E1 -13282.036,E2 -13282.036} C_VEL
LIN {X 0,Y 355.946,Z 376.149,A -85,B 0,C 180,E1 -13283.258,E2 -13283.258} C_VEL
LIN {X 0,Y 354.905,Z 376.275,A -85,B 0,C 180,E1 -13284.204,E2 -13284.204} C_VEL
LIN {X 0,Y 354.817,Z 376.286,A -85,B 0,C 180,E1 -13284.524,E2 -13284.524} C_VEL
LIN {X 0,Y 355.014,Z 376.439,A -85,B 0,C 180,E1 -13288.698,E2 -13288.698} C_VEL
LIN {X 0,Y 355.103,Z 379.537,A -85,B 0,C 180,E1 -13290.555,E2 -13290.555} C_VEL
LIN {X 0,Y 354.742,Z 385.624,A -85,B 0,C 180,E1 -13294.16,E2 -13294.16} C_VEL
LIN {X 0,Y 354.401,Z 392.036,A -85,B 0,C 180,E1 -13297.865,E2 -13297.865} C_VEL
LIN {X 0,Y 354.217,Z 397.36,A -85,B 0,C 180,E1 -13300.89,E2 -13300.89} C_VEL
LIN {X 0,Y 354.012,Z 403.759,A -85,B 0,C 180,E1 -13304.454,E2 -13304.454} C_VEL
LIN {X 0,Y 353.846,Z 410.216,A -85,B 0,C 180,E1 -13307.963,E2 -13307.963} C_VEL
LIN {X 0,Y 353.849,Z 411.137,A -85,B 0,C 180,E1 -13308.399,E2 -13308.399} C_VEL
LIN {X 0,Y 355.117,Z 422.035,A -85,B 0,C 180,E1 -13309.091,E2 -13309.091} C_VEL
LIN {X 0,Y 355.816,Z 428.556,A -85,B 0,C 180,E1 -13309.617,E2 -13309.617} C_VEL
LIN {X 0,Y 355.336,Z 438.762,A -85,B 0,C 180,E1 -13310.609,E2 -13310.609} C_VEL
LIN {X 0,Y 354.925,Z 447.783,A -85,B 0,C 180,E1 -13311.746,E2 -13311.746} C_VEL
LIN {X 0,Y 354.733,Z 455.279,A -85,B 0,C 180,E1 -13312.943,E2 -13312.943} C_VEL
LIN {X 0,Y 354.397,Z 462.071,A -85,B 0,C 180,E1 -13314.309,E2 -13314.309} C_VEL
LIN {X 0,Y 354.225,Z 466.582,A -85,B 0,C 180,E1 -13315.448,E2 -13315.448} C_VEL
LIN {X 0,Y 354.008,Z 470.213,A -85,B 0,C 180,E1 -13316.586,E2 -13316.586} C_VEL
LIN {X 0,Y 353.813,Z 474.19,A -85,B 0,C 180,E1 -13318.293,E2 -13318.293} C_VEL
LIN {X 0,Y 353.805,Z 476.575,A -85,B 0,C 180,E1 -13320,E2 -13320} C_VEL
LIN {X 0,Y 353.873,Z 477.329,A -85,B 0,C 180,E1 -13321.138,E2 -13321.138} C_VEL
LIN {X 0,Y 354.036,Z 477.421,A -85,B 0,C 180,E1 -13322.275,E2 -13322.275} C_VEL
LIN {X 0,Y 354.328,Z 476.867,A -85,B 0,C 180,E1 -13323.411,E2 -13323.411} C_VEL
LIN {X 0,Y 354.779,Z 475.656,A -85,B 0,C 180,E1 -13324.545,E2 -13324.545} C_VEL
LIN {X 0,Y 355.596,Z 472.579,A -85,B 0,C 180,E1 -13326.241,E2 -13326.241} C_VEL
LIN {X 0,Y 356.471,Z 467.876,A -85,B 0,C 180,E1 -13327.933,E2 -13327.933} C_VEL
LIN {X 0,Y 357.404,Z 462.547,A -85,B 0,C 180,E1 -13329.336,E2 -13329.336} C_VEL
LIN {X 0,Y 358.555,Z 455.685,A -85,B 0,C 180,E1 -13330.732,E2 -13330.732} C_VEL
LIN {X 0,Y 359.822,Z 447.27,A -85,B 0,C 180,E1 -13332.057,E2 -13332.057} C_VEL
LIN {X 0,Y 360.758,Z 437.881,A -85,B 0,C 180,E1 -13333.233,E2 -13333.233} C_VEL
LIN {X 0,Y 359.036,Z 427.919,A -85,B 0,C 180,E1 -13334.452,E2 -13334.452} C_VEL
LIN {X 0,Y 356.311,Z 418.779,A -85,B 0,C 180,E1 -13335.484,E2 -13335.484} C_VEL
LIN {X 0,Y 355.548,Z 416.278,A -85,B 0,C 180,E1 -13335.757,E2 -13335.757} C_VEL
LIN {X 0,Y 356.166,Z 410.777,A -85,B 0,C 180,E1 -13339.6,E2 -13339.6} C_VEL
LIN {X 0,Y 356.809,Z 406.017,A -85,B 0,C 180,E1 -13343.2,E2 -13343.2} C_VEL
LIN {X 0,Y 357.385,Z 403.003,A -85,B 0,C 180,E1 -13345.635,E2 -13345.635} C_VEL
LIN {X 0,Y 358.04,Z 400.218,A -85,B 0,C 180,E1 -13348.106,E2 -13348.106} C_VEL
LIN {X 0,Y 358.586,Z 397.649,A -85,B 0,C 180,E1 -13350.636,E2 -13350.636} C_VEL
LIN {X 0,Y 358.763,Z 395.539,A -85,B 0,C 180,E1 -13353.265,E2 -13353.265} C_VEL
LIN {X 0,Y 358.721,Z 393.919,A -85,B 0,C 180,E1 -13355.998,E2 -13355.998} C_VEL
LIN {X 0,Y 358.702,Z 392.917,A -85,B 0,C 180,E1 -13358.827,E2 -13358.827} C_VEL
LIN {X 0,Y 358.796,Z 392.646,A -85,B 0,C 180,E1 -13361.898,E2 -13361.898} C_VEL
LIN {X 0,Y 359.046,Z 393.282,A -85,B 0,C 180,E1 -13364.803,E2 -13364.803} C_VEL
LIN {X 0,Y 359.538,Z 395.061,A -85,B 0,C 180,E1 -13367.97,E2 -13367.97} C_VEL
LIN {X 0,Y 359.933,Z 396.71,A -85,B 0,C 180,E1 -13369.882,E2 -13369.882} C_VEL
LIN {X 0,Y 360.781,Z 400.337,A -85,B 0,C 180,E1 -13373.004,E2 -13373.004} C_VEL
LIN {X 0,Y 361.783,Z 404.416,A -85,B 0,C 180,E1 -13375.712,E2 -13375.712} C_VEL
LIN {X 0,Y 362.593,Z 409.719,A -85,B 0,C 180,E1 -13378.522,E2 -13378.522} C_VEL
LIN {X 0,Y 362.34,Z 412.489,A -85,B 0,C 180,E1 -13379.715,E2 -13379.715} C_VEL
LIN {X 0,Y 359.743,Z 422.177,A -85,B 0,C 180,E1 -13383.299,E2 -13383.299} C_VEL
LIN {X 0,Y 357.463,Z 434.138,A -85,B 0,C 180,E1 -13387.315,E2 -13387.315} C_VEL
LIN {X 0,Y 356.732,Z 439.38,A -85,B 0,C 180,E1 -13388.928,E2 -13388.928} C_VEL
LIN {X 0,Y 359.178,Z 451.724,A -85,B 0,C 180,E1 -13389.702,E2 -13389.702} C_VEL
LIN {X 0,Y 360.252,Z 463.13,A -85,B 0,C 180,E1 -13390.498,E2 -13390.498} C_VEL
LIN {X 0,Y 360.186,Z 475.636,A -85,B 0,C 180,E1 -13391.514,E2 -13391.514} C_VEL
LIN {X 0,Y 358.87,Z 487.227,A -85,B 0,C 180,E1 -13392.623,E2 -13392.623} C_VEL
LIN {X 0,Y 357.511,Z 497.622,A -85,B 0,C 180,E1 -13393.878,E2 -13393.878} C_VEL
LIN {X 0,Y 356.222,Z 507.548,A -85,B 0,C 180,E1 -13395.361,E2 -13395.361} C_VEL
LIN {X 0,Y 355.247,Z 515.618,A -85,B 0,C 180,E1 -13396.849,E2 -13396.849} C_VEL
LIN {X 0,Y 354.378,Z 523.172,A -85,B 0,C 180,E1 -13398.561,E2 -13398.561} C_VEL
LIN {X 0,Y 353.883,Z 529.289,A -85,B 0,C 180,E1 -13400.281,E2 -13400.281} C_VEL
LIN {X 0,Y 353.616,Z 534.139,A -85,B 0,C 180,E1 -13402.003,E2 -13402.003} C_VEL
LIN {X 0,Y 353.558,Z 537.751,A -85,B 0,C 180,E1 -13403.668,E2 -13403.668} C_VEL
LIN {X 0,Y 353.532,Z 540.513,A -85,B 0,C 180,E1 -13405.439,E2 -13405.439} C_VEL
LIN {X 0,Y 353.655,Z 541.718,A -85,B 0,C 180,E1 -13406.582,E2 -13406.582} C_VEL
LIN {X 0,Y 353.758,Z 542.509,A -85,B 0,C 180,E1 -13407.723,E2 -13407.723} C_VEL
LIN {X 0,Y 353.783,Z 542.869,A -85,B 0,C 180,E1 -13408.862,E2 -13408.862} C_VEL
LIN {X 0,Y 353.747,Z 542.742,A -85,B 0,C 180,E1 -13410,E2 -13410} C_VEL
LIN {X 0,Y 353.786,Z 542.205,A -85,B 0,C 180,E1 -13411.138,E2 -13411.138} C_VEL
LIN {X 0,Y 353.89,Z 541.243,A -85,B 0,C 180,E1 -13412.276,E2 -13412.276} C_VEL
LIN {X 0,Y 353.787,Z 539.751,A -85,B 0,C 180,E1 -13413.416,E2 -13413.416} C_VEL
LIN {X 0,Y 353.67,Z 536.632,A -85,B 0,C 180,E1 -13415.13,E2 -13415.13} C_VEL
LIN {X 0,Y 353.715,Z 532.349,A -85,B 0,C 180,E1 -13416.847,E2 -13416.847} C_VEL
LIN {X 0,Y 353.826,Z 526.757,A -85,B 0,C 180,E1 -13418.567,E2 -13418.567} C_VEL
LIN {X 0,Y 354.051,Z 519.566,A -85,B 0,C 180,E1 -13420.291,E2 -13420.291} C_VEL
LIN {X 0,Y 354.577,Z 510.537,A -85,B 0,C 180,E1 -13422.012,E2 -13422.012} C_VEL
LIN {X 0,Y 355.2,Z 501.05,A -85,B 0,C 180,E1 -13423.443,E2 -13423.443} C_VEL
LIN {X 0,Y 355.895,Z 490.62,A -85,B 0,C 180,E1 -13424.713,E2 -13424.713} C_VEL
LIN {X 0,Y 356.53,Z 480.151,A -85,B 0,C 180,E1 -13425.726,E2 -13425.726} C_VEL
LIN {X 0,Y 356.909,Z 469.871,A -85,B 0,C 180,E1 -13426.516,E2 -13426.516} C_VEL
LIN {X 0,Y 355.99,Z 457.19,A -85,B 0,C 180,E1 -13427.28,E2 -13427.28} C_VEL
LIN {X 0,Y 355.09,Z 444.957,A -85,B 0,C 180,E1 -13427.797,E2 -13427.797} C_VEL
LIN {X 0,Y 354.879,Z 441.341,A -85,B 0,C 180,E1 -13427.946,E2 -13427.946} C_VEL
LIN {X 0,Y 356.307,Z 426.355,A -85,B 0,C 180,E1 -13432.315,E2 -13432.315} C_VEL
LIN {X 0,Y 358.059,Z 412.112,A -85,B 0,C 180,E1 -13436.522,E2 -13436.522} C_VEL
LIN {X 0,Y 359.645,Z 400.915,A -85,B 0,C 180,E1 -13439.888,E2 -13439.888} C_VEL
LIN {X 0,Y 359.07,Z 396.687,A -85,B 0,C 180,E1 -13441.243,E2 -13441.243} C_VEL
LIN {X 0,Y 356.826,Z 385.966,A -85,B 0,C 180,E1 -13444.832,E2 -13444.832} C_VEL
LIN {X 0,Y 354.865,Z 376.28,A -85,B 0,C 180,E1 -13448.326,E2 -13448.326} C_VEL
LIN {X 0,Y 354.795,Z 376.292,A -85,B 0,C 180,E1 -13452.337,E2 -13452.337} C_VEL
LIN {X 0,Y 354.792,Z 376.289,A -85,B 0,C 180,E1 -13455.489,E2 -13455.489} C_VEL
LIN {X 0,Y 354.807,Z 376.286,A -85,B 0,C 180,E1 -13459.182,E2 -13459.182} C_VEL
LIN {X 0,Y 354.809,Z 376.289,A -85,B 0,C 180,E1 -13462.402,E2 -13462.402} C_VEL
LIN {X 0,Y 354.813,Z 376.286,A -85,B 0,C 180,E1 -13464.941,E2 -13464.941} C_VEL
LIN {X 0,Y 354.794,Z 376.29,A -85,B 0,C 180,E1 -13468.405,E2 -13468.405} C_VEL
LIN {X 0,Y 354.847,Z 376.283,A -85,B 0,C 180,E1 -13471.619,E2 -13471.619} C_VEL
LIN {X 0,Y 354.9,Z 376.278,A -85,B 0,C 180,E1 -13474.173,E2 -13474.173} C_VEL
LIN {X 0,Y 354.835,Z 376.287,A -85,B 0,C 180,E1 -13477.894,E2 -13477.894} C_VEL
LIN {X 0,Y 354.923,Z 376.276,A -85,B 0,C 180,E1 -13481.891,E2 -13481.891} C_VEL
LIN {X 0,Y 354.943,Z 376.273,A -85,B 0,C 180,E1 -13485.981,E2 -13485.981} C_VEL
LIN {X 0,Y 354.979,Z 376.27,A -85,B 0,C 180,E1 -13489.736,E2 -13489.736} C_VEL
LIN {X 0,Y 355.115,Z 376.25,A -85,B 0,C 180,E1 -13492.037,E2 -13492.037} C_VEL
LIN {X 0,Y 355.094,Z 376.251,A -85,B 0,C 180,E1 -13494.321,E2 -13494.321} C_VEL
LIN {X 0,Y 355.247,Z 376.236,A -85,B 0,C 180,E1 -13497.732,E2 -13497.732} C_VEL
LIN {X 0,Y 355.399,Z 376.214,A -85,B 0,C 180,E1 -13500,E2 -13500} C_VEL
LIN {X 0,Y 355.245,Z 376.232,A -85,B 0,C 180,E1 -13502.268,E2 -13502.268} C_VEL
LIN {X 0,Y 355.139,Z 376.246,A -85,B 0,C 180,E1 -13506.819,E2 -13506.819} C_VEL
LIN {X 0,Y 355.018,Z 376.264,A -85,B 0,C 180,E1 -13509.112,E2 -13509.112} C_VEL
LIN {X 0,Y 354.927,Z 376.272,A -85,B 0,C 180,E1 -13512.581,E2 -13512.581} C_VEL
LIN {X 0,Y 354.891,Z 376.275,A -85,B 0,C 180,E1 -13516.096,E2 -13516.096} C_VEL
LIN {X 0,Y 354.902,Z 376.275,A -85,B 0,C 180,E1 -13518.472,E2 -13518.472} C_VEL
LIN {X 0,Y 354.835,Z 376.283,A -85,B 0,C 180,E1 -13522.106,E2 -13522.106} C_VEL
LIN {X 0,Y 354.9,Z 376.274,A -85,B 0,C 180,E1 -13525.827,E2 -13525.827} C_VEL
LIN {X 0,Y 354.854,Z 376.281,A -85,B 0,C 180,E1 -13529.679,E2 -13529.679} C_VEL
LIN {X 0,Y 354.806,Z 376.287,A -85,B 0,C 180,E1 -13533.702,E2 -13533.702} C_VEL
LIN {X 0,Y 354.8,Z 376.289,A -85,B 0,C 180,E1 -13536.459,E2 -13536.459} C_VEL
LIN {X 0,Y 354.824,Z 376.285,A -85,B 0,C 180,E1 -13539.424,E2 -13539.424} C_VEL
LIN {X 0,Y 354.789,Z 376.293,A -85,B 0,C 180,E1 -13542.868,E2 -13542.868} C_VEL
LIN {X 0,Y 354.77,Z 376.292,A -85,B 0,C 180,E1 -13546.104,E2 -13546.104} C_VEL
LIN {X 0,Y 354.79,Z 376.29,A -85,B 0,C 180,E1 -13549.18,E2 -13549.18} C_VEL
LIN {X 0,Y 354.813,Z 376.289,A -85,B 0,C 180,E1 -13552.402,E2 -13552.402} C_VEL
LIN {X 0,Y 354.813,Z 376.288,A -85,B 0,C 180,E1 -13554.941,E2 -13554.941} C_VEL
LIN {X 0,Y 354.795,Z 376.292,A -85,B 0,C 180,E1 -13558.405,E2 -13558.405} C_VEL
LIN {X 0,Y 354.848,Z 376.281,A -85,B 0,C 180,E1 -13561.619,E2 -13561.619} C_VEL
LIN {X 0,Y 354.901,Z 376.278,A -85,B 0,C 180,E1 -13564.173,E2 -13564.173} C_VEL
LIN {X 0,Y 354.841,Z 376.284,A -85,B 0,C 180,E1 -13567.895,E2 -13567.895} C_VEL
LIN {X 0,Y 354.925,Z 376.273,A -85,B 0,C 180,E1 -13571.891,E2 -13571.891} C_VEL
LIN {X 0,Y 354.945,Z 376.273,A -85,B 0,C 180,E1 -13575.981,E2 -13575.981} C_VEL
LIN {X 0,Y 354.982,Z 376.266,A -85,B 0,C 180,E1 -13579.736,E2 -13579.736} C_VEL
LIN {X 0,Y 355.128,Z 376.246,A -85,B 0,C 180,E1 -13583.181,E2 -13583.181} C_VEL
LIN {X 0,Y 355.247,Z 376.235,A -85,B 0,C 180,E1 -13587.733,E2 -13587.733} C_VEL
LIN {X 0,Y 355.401,Z 376.217,A -85,B 0,C 180,E1 -13590,E2 -13590} C_VEL
LIN {X 0,Y 355.247,Z 376.234,A -85,B 0,C 180,E1 -13592.268,E2 -13592.268} C_VEL
LIN {X 0,Y 355.127,Z 376.246,A -85,B 0,C 180,E1 -13596.82,E2 -13596.82} C_VEL
LIN {X 0,Y 354.981,Z 376.267,A -85,B 0,C 180,E1 -13600.264,E2 -13600.264} C_VEL
LIN {X 0,Y 354.946,Z 376.272,A -85,B 0,C 180,E1 -13604.019,E2 -13604.019} C_VEL
LIN {X 0,Y 354.926,Z 376.274,A -85,B 0,C 180,E1 -13608.109,E2 -13608.109} C_VEL
LIN {X 0,Y 354.837,Z 376.284,A -85,B 0,C 180,E1 -13612.106,E2 -13612.106} C_VEL
LIN {X 0,Y 354.902,Z 376.278,A -85,B 0,C 180,E1 -13615.828,E2 -13615.828} C_VEL
LIN {X 0,Y 354.82,Z 376.289,A -85,B 0,C 180,E1 -13619.682,E2 -13619.682} C_VEL
LIN {X 0,Y 354.809,Z 376.289,A -85,B 0,C 180,E1 -13623.702,E2 -13623.702} C_VEL
LIN {X 0,Y 354.803,Z 376.286,A -85,B 0,C 180,E1 -13626.459,E2 -13626.459} C_VEL
LIN {X 0,Y 354.827,Z 376.288,A -85,B 0,C 180,E1 -13629.424,E2 -13629.424} C_VEL
LIN {X 0,Y 354.791,Z 376.291,A -85,B 0,C 180,E1 -13632.867,E2 -13632.867} C_VEL
LIN {X 0,Y 354.783,Z 376.289,A -85,B 0,C 180,E1 -13636.106,E2 -13636.106} C_VEL
LIN {X 0,Y 354.78,Z 376.291,A -85,B 0,C 180,E1 -13639.595,E2 -13639.595} C_VEL
